(* CODESYS project SingleElevator_final.project

Project tree, tasks and I/O mapping:
  Device : CODESYS Control Win V3, 3S - Smart Software Solutions GmbH, version 3.5.15.40
    application Application
      libraries: Standard, * (System)
      task MainTask (cyclic, interval 100 ms, priority 1) calls Simulation, GA_collector, Policy
      task VISU_TASK (cyclic, interval 100 ms, priority 31) calls VisuElems.Visu_Prg
      global variables GVL
      visualisation Visualization
      program Simulation [ST]
      GAs/
        function block Door_module [SFC]: ready_active, busy_active, op_complete_active, reset_done_active, Init_active
        function block Cardinal [SFC]: Lights_active, Busy_active, Ready_active, Save_Arrays_active, Init_active, Cancel_call_active
        function block Moves_module [SFC]: G_floor_Problem_active, Stop_Op_Doors_down_active, Ready_active, Busy_active, Closing_Doors_active, Closing_Doors_exit, Init_active, Stop_Op_Doors_down_exit, Slow_d_active, Stop_Op_Doors_up_active, Slow_u_active, Fast_u_active, Stop_Op_Doors_up_exit, Check_Ramp_u_active, Check_Deck_u_active, Fast_d_active, Check_Ramp_d_active, Check_Deck_d_active, Stop_u_active, Stop_d_active, Errors_d_active, Errors_u_active, Homing_0_active, Homing_0_exit, Homing_1_active, Homing_2_active, Homing_3_active, Homing_3_exit, Exception_2_active, Exception_3_active, Exception_3_exit
      program GA_collector [FBD]
      program Policy [SFC]: Start_Cardinal_active, Error_routines_active, Start_Homing_active, Start_What_active, _aFinish_routine_active
  text list GlobalTextList
*)

// Device/Application/GVL
//{attribute 'qualified_only'}
VAR_GLOBAL
(* Elevator managing variables*)
	Open: BOOL;				(* Sensor: the door is fully open*)
	Closed: BOOL;			(* Sensor: the door is fully closed*)
	LimitDown: BOOL;		(* Sensor: lower limit sensor, if TRUE the lift has reached the lower limit*)
	LimitUp: BOOL;			(* Sensor: upper limit sensor, if TRUE the lift has reached the upper limit*)
	DeckSensor: BOOL;		(* Sensor: if TRUE the cab is in proximity of a deck*)
	RampSensor: BOOL;		(* Sensor: if TRUE the cab is in proximity of a ramp*)
	Presence :BOOL; 		(* Sensor: if TRUE something blocks the door photocell*)
	Emergency: BOOL;		(* Input: if TRUE the emergency button has been pressed*)

	Closing: BOOL;			(* Actuator: if TRUE the door starts closing*)
	Opening: BOOL;			(* Actuator: the door starts opening*)
	Motor_on: BOOL;			(* Actuator: if TRUE the lift pulley motor start moving*)
	Up: BOOL;				(* Actuator parameter: if TRUE the lift moves upward, downward otherwise*)
	Vel: BOOL;				(* Actuator parameter: motor speed, if TRUE high speed, low speed otherwise*)
	

	Current: INT;  			(* Visualization: variable used to storage the current deck*)
    Destination: INT;		(* Visualization: variable used to storage the the destination deck*)
	EmergencyVis: BOOL; 	(* Visualization: if TRUE the emergency light is turned on*)


	
	
	InitialDeck: INT := 1;	(* Only for simulation: variable used to define the initial deck*)
	InitCycle: BOOL := FALSE;(* Only for simulation: used to execute the instruction at the first cycle*)
	Height: INT;			(* Only for simulation: elevator height*)
	DeckRest: INT;        	(* Only for simulation: division rest for generating deck sensor*)
	Memory: INT;
	RampRest: INT;			(* Only for simulation: division rest for generating the ramp position*)
	MemoryR: INT;
	Door: INT;				(* Only for simulation: to visualize the closing of the door*)
	Displacement: INT;		(* Only for simulation: lift displacement, dependent on the motor speed*)

 (*Inputs: internal panel variables*)
	PG: BOOL;
	P1: BOOL;
	P2: BOOL;
	P3: BOOL;
	P4: BOOL;
	P5: BOOL;
	P6: BOOL;
	P7: BOOL;
	
	(*Inputs: external panel variables*)
	UpDeckG: BOOL;
	UpDeck1: BOOL;
	UpDeck2: BOOL;
	UpDeck3: BOOL;
	UpDeck4: BOOL;
	UpDeck5: BOOL;
	UpDeck6: BOOL;
	DownDeck7: BOOL;
	DownDeck6: BOOL;
	DownDeck5: BOOL;
	DownDeck4: BOOL;
	DownDeck3: BOOL;
	DownDeck2: BOOL;
	DownDeck1: BOOL;

(*Visualization: internal panel variables used to turn on the LED*)
	PGVis: BOOL;
	P1Vis: BOOL;
	P2Vis: BOOL;
	P3Vis: BOOL;
	P4Vis: BOOL;
	P5Vis: BOOL;
	P6Vis: BOOL;
	P7Vis: BOOL;

(*Visualization: external panel variables used to turn on the LED*)
	UpDeckGVis: BOOL;
	UpDeck1Vis: BOOL;
	UpDeck2Vis: BOOL;
	UpDeck3Vis: BOOL;
	UpDeck4Vis: BOOL;
	UpDeck5Vis: BOOL;
	UpDeck6Vis: BOOL;
	DownDeck7Vis: BOOL;
	DownDeck6Vis: BOOL;
	DownDeck5Vis: BOOL;
	DownDeck4Vis: BOOL;
	DownDeck3Vis: BOOL;
	DownDeck2Vis: BOOL;
	DownDeck1Vis: BOOL;

(*Only for simulation: variables used to simulate the fault on deck sensor*)
	SensorG: BOOL;				(* if TRUE the magnetic information for deck G is lost and the deck sensor cannot become TRUE*)
	Sensor1: BOOL;				(* if TRUE the magnetic information for deck 1 is lost and the deck sensor cannot become TRUE*)
	Sensor2: BOOL;
	Sensor3: BOOL;
	Sensor4: BOOL;
	Sensor5: BOOL;
	Sensor6: BOOL;
	Sensor7: BOOL;
	FaultSensorAlarm: BOOL; 	(* Visulaization: if TRUE alerts the user of a deck sensor fault*)

(*Only for simulation: variables used to simulate the fault on ramp sensor*)
	RampGUp: BOOL;
	Ramp1Down: BOOL;
	Ramp1Up:BOOL;
	Ramp2Down: BOOL;
	Ramp2Up:BOOL;
	Ramp3Down: BOOL;
	Ramp3Up:BOOL;
	Ramp4Down: BOOL;
	Ramp4Up:BOOL;
	Ramp5Down: BOOL;
	Ramp5Up:BOOL;
	Ramp6Down: BOOL;
	Ramp6Up:BOOL;
	Ramp7Down: BOOL;
	FaultRampAlarm: BOOL; 		(* Visulaization: if TRUE alerts the user of a ramp sensor fault*)
	SensorGOK: BOOL;
	Sensor1OK: BOOL;
	Sensor2OK: BOOL;
	Sensor6OK: BOOL;
	Sensor3OK: BOOL;
	Sensor4OK: BOOL;
	Sensor5OK: BOOL;
	Sensor7OK: BOOL;
	RampGUpOK: BOOL;
	Ramp1DownOK: BOOL;
	Ramp1UpOK: BOOL;
	Ramp2DownOK: BOOL;
	Ramp2UpOK: BOOL;
	Ramp3DownOK: BOOL;
	Ramp3UpOK: BOOL;
	Ramp4DownOK: BOOL;
	Ramp4UpOK: BOOL;
	Ramp5DownOK: BOOL;
	Ramp5UpOK: BOOL;
	Ramp6DownOK: BOOL;
	Ramp6UpOK: BOOL;
	Ramp7DownOK: BOOL;
	Ramp7UpOK: BOOL;
	
	//var aggiunte da me
	array_dest_up_onfly: ARRAY[0..7] OF INT;
	array_dest_up_stored: ARRAY[0..7] OF INT;
	
	array_dest_down_onfly: ARRAY[0..7] OF INT;
	array_dest_down_stored: ARRAY[0..7] OF INT;
	
	served_up: BOOL; // flag di fine servizio per movimento up
	served_down: BOOL; // flag di fine servizio per movimento down
	dest_target_up: INT; //destinazioen target up
	dest_target_down: INT; //destinazione target down
	enable_target_up_down: BOOL;	
	G_floor_problem: BOOL;
	
	//Istanze dei GA
	door_module_0: Door_module;
	Cardinal_0: Cardinal;
	Moves_module_0: Moves_module;

END_VAR

// Device/Application/Simulation
PROGRAM Simulation
VAR
END_VAR

(* Initial position of the cab inside the hoistway. It is executed only at the first cycle.  *)
IF NOT GVL.InitCycle THEN
			GVL.InitCycle := TRUE ;
			GVL.Height := 20 * GVL.InitialDeck;
		    GVL.Door := 0;
			GVL.Current := GVL.Height / 20;
END_IF;

(* Elevator management, these instructions are executed each cycle time*)

(* Elevator door control. *)
IF GVL.Closing THEN
	GVL.Door := GVL.Door + 1;		(*Closing door management*)
	GVL.Open := FALSE;
END_IF

IF GVL.Door >= 60 THEN						(* Closed door limit*)
	GVL.Closed := TRUE;
END_IF

IF GVL.Opening THEN
	GVL.Door := GVL.Door - 1; 	(* Opening door management*)
	GVL.Closed := FALSE;
END_IF

IF GVL.Door <= 0 THEN							(* Open door limit*)
	GVL.Open := TRUE;
END_IF


(* Maximum and minimum management in the door simulation*)
IF GVL.Door < 0 THEN
	 GVL.Door := 0;
END_IF

IF GVL.Door > 60 THEN
	GVL.Door := 60;
END_IF


(* Control of the cab position inside the hostway. *)
(* Displacement definition for graphic visualization*)
IF GVL.Vel THEN 
	GVL.Displacement := 2;
ELSE 
	GVL.Displacement := 1;
END_IF


(* Height modification relying on direction and speed*)
IF GVL.Motor_on AND GVL.Up THEN
	GVL.Height := GVL.Height + GVL.Displacement;
	GVL.LimitDown := FALSE;
END_IF

IF GVL.Motor_on AND NOT GVL.Up THEN
	GVL.Height := GVL.Height - GVL.Displacement;
	GVL.LimitUp := FALSE;
END_IF


(* Limits for visualization*)
IF GVL.Height < -20 THEN
	GVL.Height := -20;
END_IF

IF GVL.Height > 160 THEN
	GVL.Height := 160;
END_IF

(* Limit sensors management*)
IF GVL.Height <= -10 THEN
	GVL.LimitDown := TRUE;
END_IF

IF GVL.Height >= 150 THEN
	 GVL.LimitUp := TRUE;
END_IF


(*-------------------------------------------------------------------*)
(*  Fault Management (Deck and Ramp Sensors)   *)
(*-------------------------------------------------------------------*)
(* Deck Sensor*)
(* Range of value where the deck sensor is active*)
IF ((GVL.Height >= -1) AND (GVL.Height <= 1)) THEN
	GVL.SensorGOK := TRUE;
ELSE  
	GVL.SensorGOK := FALSE;
END_IF

IF ((GVL.Height >= 20-1) AND (GVL.Height <= 20+1)) THEN
	GVL.Sensor1OK := TRUE;
ELSE  
	GVL.Sensor1OK := FALSE;
END_IF

IF ((GVL.Height >= 40-1) AND (GVL.Height <= 40+1)) THEN
	GVL.Sensor2OK := TRUE;
ELSE  
	GVL.Sensor2OK := FALSE;
END_IF

IF ((GVL.Height >= 60-1) AND (GVL.Height <= 60+1)) THEN
	GVL.Sensor3OK := TRUE;
ELSE  
	GVL.Sensor3OK := FALSE;
END_IF

IF ((GVL.Height >= 80-1) AND (GVL.Height <= 80+1)) THEN
	GVL.Sensor4OK := TRUE;
ELSE  
	GVL.Sensor4OK := FALSE;
END_IF

IF ((GVL.Height >= 100-1) AND (GVL.Height <= 100+1)) THEN
	GVL.Sensor5OK := TRUE;
ELSE   
	GVL.Sensor5OK := FALSE;
END_IF

IF ((GVL.Height >= 120-1) AND (GVL.Height <= 120+1)) THEN
	GVL.Sensor6OK := TRUE;
ELSE  
	GVL.Sensor6OK := FALSE;
END_IF

IF ((GVL.Height >= 140-1) AND (GVL.Height <= 140+1)) THEN
	GVL.Sensor7OK := TRUE;
ELSE  
	GVL.Sensor7OK := FALSE;
END_IF

GVL.DeckSensor := (GVL.SensorGOK AND NOT GVL.SensorG) OR
				    (GVL.Sensor1OK AND NOT GVL.Sensor1) OR
				    (GVL.Sensor2OK AND NOT GVL.Sensor2) OR
				    (GVL.Sensor3OK AND NOT GVL.Sensor3) OR
				    (GVL.Sensor4OK AND NOT GVL.Sensor4) OR
				    (GVL.Sensor5OK AND NOT GVL.Sensor5) OR
				    (GVL.Sensor6OK AND NOT GVL.Sensor6) OR
				    (GVL.Sensor7OK AND NOT GVL.Sensor7);

(* Ramp Sensor*)
(* Range of value where the ramp sensor is active*)
IF ((GVL.Height >= 5-1) AND (GVL.Height <= 5+1)) THEN
	GVL.RampGUpOK := TRUE;
ELSE 
	GVL.RampGUpOK := FALSE;
END_IF

(* Ramp close to deck 1*)
IF ((GVL.Height >= 15-1) AND (GVL.Height <= 15+1)) THEN
	GVL.Ramp1DownOK := TRUE;
ELSE 
	GVL.Ramp1DownOK := FALSE;
END_IF

IF ((GVL.Height >= 25-1) AND (GVL.Height <= 25+1)) THEN
	GVL.Ramp1UpOK := TRUE;
ELSE 
	GVL.Ramp1UpOK := FALSE;
END_IF

(* Ramp close to deck 2*)
IF ((GVL.Height >= 35-1) AND (GVL.Height <= 35+1)) THEN
	GVL.Ramp2DownOK := TRUE;
ELSE 
	GVL.Ramp2DownOK := FALSE;
END_IF

IF ((GVL.Height >= 45-1) AND (GVL.Height <= 45+1)) THEN
	GVL.Ramp2UpOK := TRUE;
ELSE 
	GVL.Ramp2UpOK := FALSE;
END_IF

(*Ramp close to deck  3*)
IF ((GVL.Height >= 55-1) AND (GVL.Height <= 55+1)) THEN
	GVL.Ramp3DownOK := TRUE;
ELSE 
	GVL.Ramp3DownOK := FALSE;
END_IF

IF ((GVL.Height >= 65-1) AND (GVL.Height <= 65+1)) THEN
	GVL.Ramp3UpOK := TRUE;
ELSE 
	GVL.Ramp3UpOK := FALSE;
END_IF

(* Ramp close to deck  4*)
IF ((GVL.Height >= 75-1) AND (GVL.Height <= 75+1)) THEN
	GVL.Ramp4DownOK := TRUE;
ELSE 
	GVL.Ramp4DownOK := FALSE;
END_IF

IF ((GVL.Height >= 85-1) AND (GVL.Height <= 85+1)) THEN
	GVL.Ramp4UpOK := TRUE;
ELSE 
	GVL.Ramp4UpOK:=FALSE;
END_IF

(* Ramp close to deck  5*)
IF ((GVL.Height >= 95-1) AND (GVL.Height <= 95+1)) THEN
	GVL.Ramp5DownOK := TRUE;
ELSE 
	GVL.Ramp5DownOK := FALSE;
END_IF

IF ((GVL.Height >= 105-1) AND (GVL.Height <= 105+1)) THEN
	GVL.Ramp5UpOK := TRUE;
ELSE
	GVL.Ramp5UpOK := FALSE;
END_IF

(* Ramp close to deck  6*)
IF ((GVL.Height >= 115-1) AND (GVL.Height <= 115+1)) THEN
	GVL.Ramp6DownOK := TRUE;
ELSE 
	GVL.Ramp6DownOK := FALSE;
END_IF

IF ((GVL.Height >= 125-1) AND (GVL.Height <= 125+1)) THEN
	GVL.Ramp6UpOK := TRUE;
ELSE 
	GVL.Ramp6UpOK := FALSE;
END_IF

(* Ramp close to deck  7*)
IF ((GVL.Height >= 135-1) AND (GVL.Height <= 135+1)) THEN
	GVL.Ramp7DownOK := TRUE;
ELSE 
	GVL.Ramp7DownOK := FALSE;
END_IF

GVL.RampSensor:=(GVL.RampGUpOK AND NOT GVL.RampGUp) OR 
								(GVL.Ramp1DownOK AND NOT GVL.Ramp1Down ) OR 
								(GVL.Ramp1UpOK AND NOT GVL.Ramp1Up ) OR
								(GVL.Ramp2DownOK AND NOT GVL.Ramp2Down ) OR 
								(GVL.Ramp2UpOK AND NOT GVL.Ramp2Up ) OR
								(GVL.Ramp3DownOK AND NOT GVL.Ramp3Down ) OR
 								(GVL.Ramp3UpOK AND NOT GVL.Ramp3Up ) OR
								(GVL.Ramp4DownOK AND NOT GVL.Ramp4Down ) OR
 								(GVL.Ramp4UpOK AND NOT GVL.Ramp4Up ) OR
								(GVL.Ramp5DownOK AND NOT GVL.Ramp5Down ) OR
 								(GVL.Ramp5UpOK AND NOT GVL.Ramp5Up ) OR
								(GVL.Ramp6DownOK AND NOT GVL.Ramp6Down ) OR
								(GVL.Ramp6UpOK AND NOT GVL.Ramp6Up ) OR
								(GVL.Ramp7DownOK AND NOT GVL.Ramp7Down );

END_PROGRAM

// Device/Application/GA_collector
PROGRAM GA_collector
VAR



END_VAR

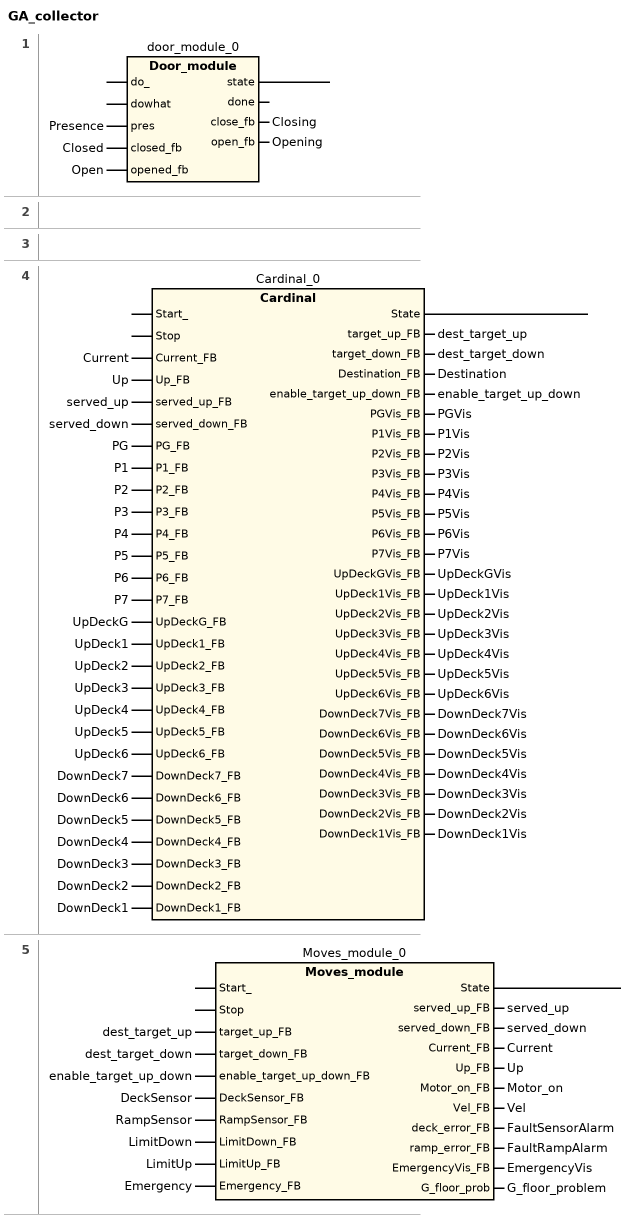
// NETWORK 1
door_module_0(
    pres := Presence,
    closed_fb := Closed,
    opened_fb := Open,
    close_fb => Closing,
    open_fb => Opening); // Door_module

// NETWORK 2

// NETWORK 3

// NETWORK 4
Cardinal_0(
    Current_FB := Current,
    Up_FB := Up,
    served_up_FB := served_up,
    served_down_FB := served_down,
    PG_FB := PG,
    P1_FB := P1,
    P2_FB := P2,
    P3_FB := P3,
    P4_FB := P4,
    P5_FB := P5,
    P6_FB := P6,
    P7_FB := P7,
    UpDeckG_FB := UpDeckG,
    UpDeck1_FB := UpDeck1,
    UpDeck2_FB := UpDeck2,
    UpDeck3_FB := UpDeck3,
    UpDeck4_FB := UpDeck4,
    UpDeck5_FB := UpDeck5,
    UpDeck6_FB := UpDeck6,
    DownDeck7_FB := DownDeck7,
    DownDeck6_FB := DownDeck6,
    DownDeck5_FB := DownDeck5,
    DownDeck4_FB := DownDeck4,
    DownDeck3_FB := DownDeck3,
    DownDeck2_FB := DownDeck2,
    DownDeck1_FB := DownDeck1,
    target_up_FB => dest_target_up,
    target_down_FB => dest_target_down,
    Destination_FB => Destination,
    enable_target_up_down_FB => enable_target_up_down,
    PGVis_FB => PGVis,
    P1Vis_FB => P1Vis,
    P2Vis_FB => P2Vis,
    P3Vis_FB => P3Vis,
    P4Vis_FB => P4Vis,
    P5Vis_FB => P5Vis,
    P6Vis_FB => P6Vis,
    P7Vis_FB => P7Vis,
    UpDeckGVis_FB => UpDeckGVis,
    UpDeck1Vis_FB => UpDeck1Vis,
    UpDeck2Vis_FB => UpDeck2Vis,
    UpDeck3Vis_FB => UpDeck3Vis,
    UpDeck4Vis_FB => UpDeck4Vis,
    UpDeck5Vis_FB => UpDeck5Vis,
    UpDeck6Vis_FB => UpDeck6Vis,
    DownDeck7Vis_FB => DownDeck7Vis,
    DownDeck6Vis_FB => DownDeck6Vis,
    DownDeck5Vis_FB => DownDeck5Vis,
    DownDeck4Vis_FB => DownDeck4Vis,
    DownDeck3Vis_FB => DownDeck3Vis,
    DownDeck2Vis_FB => DownDeck2Vis,
    DownDeck1Vis_FB => DownDeck1Vis); // Cardinal

// NETWORK 5
Moves_module_0(
    target_up_FB := dest_target_up,
    target_down_FB := dest_target_down,
    enable_target_up_down_FB := enable_target_up_down,
    DeckSensor_FB := DeckSensor,
    RampSensor_FB := RampSensor,
    LimitDown_FB := LimitDown,
    LimitUp_FB := LimitUp,
    Emergency_FB := Emergency,
    served_up_FB => served_up,
    served_down_FB => served_down,
    Current_FB => Current,
    Up_FB => Up,
    Motor_on_FB => Motor_on,
    Vel_FB => Vel,
    deck_error_FB => FaultSensorAlarm,
    ramp_error_FB => FaultRampAlarm,
    EmergencyVis_FB => EmergencyVis,
    G_floor_prob => G_floor_problem); // Moves_module

END_PROGRAM

// Device/Application/GAs/Door_module
FUNCTION_BLOCK Door_module
VAR_INPUT
	do_: BOOL;
	dowhat: STRING;
	pres: BOOL;
	closed_fb: BOOL;
	opened_fb: BOOL;
END_VAR
VAR_OUTPUT
	state: STRING;
	done: BOOL;
	close_fb: BOOL;
	open_fb: BOOL;
END_VAR
VAR
END_VAR

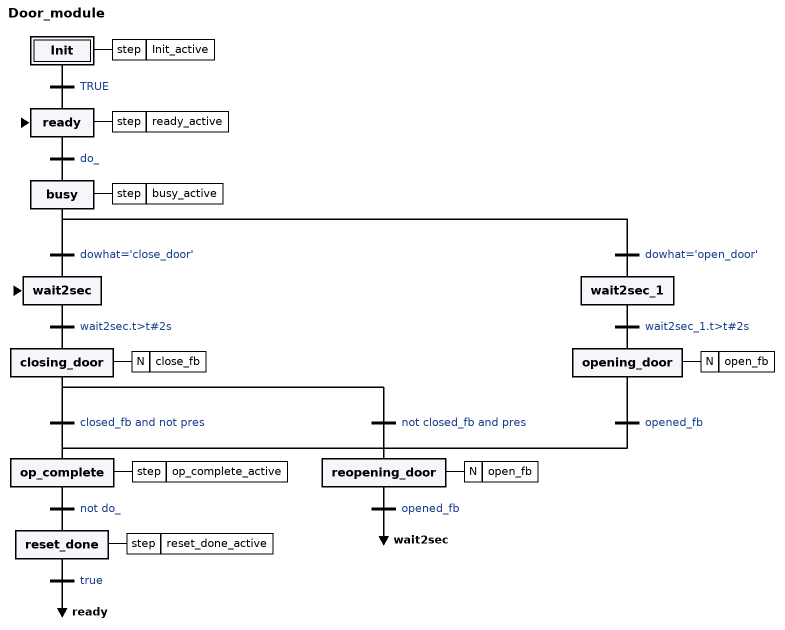
INITIAL_STEP Init:
    Init_active(N);  // step action
END_STEP
TRANSITION FROM Init TO ready
    := TRUE;
END_TRANSITION
STEP ready:
    ready_active(N);  // step action
END_STEP
TRANSITION FROM ready TO busy
    := do_;
END_TRANSITION
STEP busy:
    busy_active(N);  // step action
END_STEP
TRANSITION FROM busy TO wait2sec
    := dowhat='close_door';
END_TRANSITION
STEP wait2sec:
END_STEP
TRANSITION FROM wait2sec TO closing_door
    := wait2sec.t>t#2s;
END_TRANSITION
STEP closing_door:
    close_fb(N);
END_STEP
TRANSITION FROM closing_door TO op_complete
    := closed_fb and not pres;
END_TRANSITION
TRANSITION FROM closing_door TO reopening_door
    := not closed_fb and pres;
END_TRANSITION
STEP reopening_door:
    open_fb(N);
END_STEP
TRANSITION FROM reopening_door TO wait2sec
    := opened_fb;
END_TRANSITION
TRANSITION FROM busy TO wait2sec_1
    := dowhat='open_door';
END_TRANSITION
STEP wait2sec_1:
END_STEP
TRANSITION FROM wait2sec_1 TO opening_door
    := wait2sec_1.t>t#2s;
END_TRANSITION
STEP opening_door:
    open_fb(N);
END_STEP
TRANSITION FROM opening_door TO op_complete
    := opened_fb;
END_TRANSITION
STEP op_complete:
    op_complete_active(N);  // step action
END_STEP
TRANSITION FROM op_complete TO reset_done
    := not do_;
END_TRANSITION
STEP reset_done:
    reset_done_active(N);  // step action
END_STEP
TRANSITION FROM reset_done TO ready
    := true;
END_TRANSITION

ACTION ready_active:
state:='ready';
END_ACTION

ACTION busy_active:
state:='busy';
END_ACTION

ACTION op_complete_active:
done:=TRUE;
END_ACTION

ACTION reset_done_active:
done:=FALSE;
END_ACTION

ACTION Init_active:
//INZIALIZZAZIONE DEGLI OUTPUT DI DOOR_MODULE
done:=FALSE;
close_fb:=FALSE;
open_fb:=FALSE;
END_ACTION

END_FUNCTION_BLOCK

// Device/Application/GAs/Cardinal
FUNCTION_BLOCK Cardinal
VAR_INPUT
	
	Start_: BOOL;
	Stop: BOOL;
	Current_FB: INT; //visualizzazione piano corrente	

	Up_FB:BOOL;
	
	served_up_FB: BOOL; // flag di finito servizio del valore target_up
	served_down_FB: BOOL; // flag di finito servizio del valore target_down
	
	 (*Inputs: internal panel variables*)
	PG_FB: BOOL;
	P1_FB: BOOL;
	P2_FB: BOOL;
	P3_FB: BOOL;
	P4_FB: BOOL;
	P5_FB: BOOL;
	P6_FB: BOOL;
	P7_FB: BOOL;
	
	(*Inputs: external panel variables*)
	UpDeckG_FB: BOOL;
	UpDeck1_FB: BOOL;
	UpDeck2_FB: BOOL;
	UpDeck3_FB: BOOL;
	UpDeck4_FB: BOOL;
	UpDeck5_FB: BOOL;
	UpDeck6_FB: BOOL;
	DownDeck7_FB: BOOL;
	DownDeck6_FB: BOOL;
	DownDeck5_FB: BOOL;
	DownDeck4_FB: BOOL;
	DownDeck3_FB: BOOL;
	DownDeck2_FB: BOOL;
	DownDeck1_FB: BOOL;
END_VAR
VAR_OUTPUT
	
	State: STRING;
	
	target_up_FB: INT; // valore da dare a Dest_target_up
	target_down_FB: INT; // valore da dare a Dest_target_down
	
	Destination_FB: INT; //visualizzazione del piano destinazione
	
	enable_target_up_down_FB: BOOL; //per manovrare in moves_module il verso di percorrenza
	
(*Visualization: internal panel variables used to turn on the LED*)
	PGVis_FB: BOOL;
	P1Vis_FB: BOOL;
	P2Vis_FB: BOOL;
	P3Vis_FB: BOOL;
	P4Vis_FB: BOOL;
	P5Vis_FB: BOOL;
	P6Vis_FB: BOOL;
	P7Vis_FB: BOOL;

(*Visualization: external panel variables used to turn on the LED*)
	UpDeckGVis_FB: BOOL;
	UpDeck1Vis_FB: BOOL;
	UpDeck2Vis_FB: BOOL;
	UpDeck3Vis_FB: BOOL;
	UpDeck4Vis_FB: BOOL;
	UpDeck5Vis_FB: BOOL;
	UpDeck6Vis_FB: BOOL;
	DownDeck7Vis_FB: BOOL;
	DownDeck6Vis_FB: BOOL;
	DownDeck5Vis_FB: BOOL;
	DownDeck4Vis_FB: BOOL;
	DownDeck3Vis_FB: BOOL;
	DownDeck2Vis_FB: BOOL;
	DownDeck1Vis_FB: BOOL;
	
END_VAR
VAR
	Dest_floor: INT;//contiene variabile destinazione
	can_be_clicked: BOOL;
	up_motion: BOOL; 
	prio: INT;

	//ARRAY DELLE CHIAMATE

	array_dest_up_onfly_FB: ARRAY[0..7] OF INT;

	array_dest_up_stored_FB: ARRAY[0..7] OF INT;
	

	array_dest_down_onfly_FB: ARRAY[0..7] OF INT;

	array_dest_down_stored_FB: ARRAY[0..7] OF INT;
	
	// contatori di scorrimento per la scrittura degli array,
	sliding_index_1: INT;
	sliding_index_2: INT;
	sliding_index_3: INT;
	sliding_index_4: INT;
	
	// contatori di riordino array
	k: INT;
	i: INT;
	k_1: INT;
	i_1: INT;

	//variabili appoggio riordino array
	var1: INT;

	var1_1: INT;
	
	min_index: INT;
	min_index_1: INT;
	max_index: INT;
	max_index_1: INT;
	already_pres: BOOL;

	//contatori generici 	
	counter_calls_up_stored: INT;
	counter_calls_down_stored: INT;
	counter_calls_up_onfly: INT;
	counter_calls_down_onfly: INT;

	cont: INT;
	cancel_time: BOOL;
END_VAR

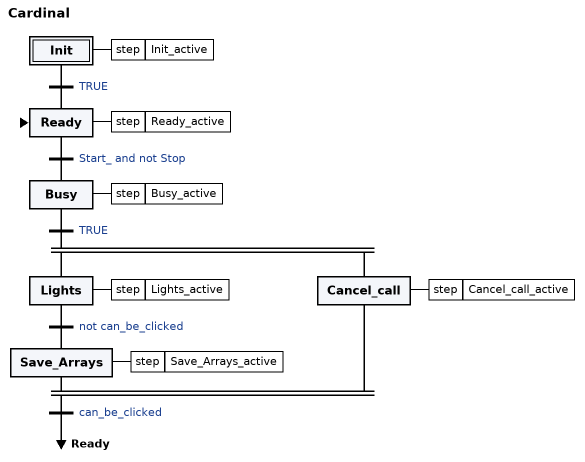
INITIAL_STEP Init:
    Init_active(N);  // step action
END_STEP
TRANSITION FROM Init TO Ready
    := TRUE;
END_TRANSITION
STEP Ready:
    Ready_active(N);  // step action
END_STEP
TRANSITION FROM Ready TO Busy
    := Start_ and not Stop;
END_TRANSITION
STEP Busy:
    Busy_active(N);  // step action
END_STEP
TRANSITION FROM Busy TO (Lights, Cancel_call)
    := TRUE;
END_TRANSITION
STEP Lights:
    Lights_active(N);  // step action
END_STEP
TRANSITION FROM Lights TO Save_Arrays
    := not can_be_clicked;
END_TRANSITION
STEP Save_Arrays:
    Save_Arrays_active(N);  // step action
END_STEP
STEP Cancel_call:
    Cancel_call_active(N);  // step action
END_STEP
TRANSITION FROM (Save_Arrays, Cancel_call) TO Ready
    := can_be_clicked;
END_TRANSITION

ACTION Lights_active:
//INTERFACCIAMENTO CON LE CHIAMATE DA PULSANTIERA INTERNA
(*
HO SCELTO DI DARE A QUESTE CHIAMATE UN 'VERSO' IN MODO DA TRATTARLE ALLO STESSO MODO DELLE CHIAMATE
DA PULSANTIERA ESTERNA, IL VERSO IN QUESTIONE DERIVA DAL FLAG up_elev_curr_FB CHE DERIVA DAL FLAG
DEL VERSO DELL'ASCENSORE IN USCITA DAL GA DI MOVIMENTO (MOVES_MODULE) CON VALORE AD INIZIO PROGRAMMA
PARI A TRUE PERCHE DOPO L'HOMING POSSO SOLO ANDARE IN ALTO. E' UN PRINCIPIO DI RETROAZIONE PERCHE A 
SUA VOLTA MOVES_MODULE LEGGERA' LE USCITE DI CARDINAL PER SAPERE LA DESTINAZIONE.
*)

//up_elev_curr_FB: FLAG IN INGRESSO AL CARDINAL E IN OUTPUT A MOVES_MODULE
//up_motion: VIENE LETTO DOPO PER SAPERE DOVE SMISTARE LE CALLS

IF PG_FB AND can_be_clicked THEN
	PGVis_FB:=TRUE;
	can_be_clicked:=FALSE;
	Dest_floor:=0;
	IF Dest_floor>Current_FB THEN
		up_motion:=TRUE;
	ELSE
		up_motion:=FALSE;
	END_IF
END_IF
IF P1_FB AND can_be_clicked THEN
	P1Vis_FB:=TRUE;
	can_be_clicked:=FALSE;
	Dest_floor:=1;
	IF Dest_floor>Current_FB THEN
		up_motion:=TRUE;
	ELSE
		up_motion:=FALSE;
	END_IF
END_IF
IF P2_FB AND can_be_clicked  THEN
	P2Vis_FB:=TRUE;
	can_be_clicked:=FALSE;
	Dest_floor:=2;
	IF Dest_floor>Current_FB THEN
		up_motion:=TRUE;
	ELSE
		up_motion:=FALSE;
	END_IF
END_IF
IF P3_FB AND can_be_clicked  THEN
	P3Vis_FB:=TRUE;
	can_be_clicked:=FALSE;
	Dest_floor:=3;
	IF Dest_floor>Current_FB THEN
		up_motion:=TRUE;
	ELSE
		up_motion:=FALSE;
	END_IF
END_IF
IF P4_FB AND can_be_clicked  THEN
	P4Vis_FB:=TRUE;
	can_be_clicked:=FALSE;
	Dest_floor:=4;
	IF Dest_floor>Current_FB THEN
		up_motion:=TRUE;
	ELSE
		up_motion:=FALSE;
	END_IF
END_IF
IF P5_FB AND can_be_clicked  THEN
	P5Vis_FB:=TRUE;
	can_be_clicked:=FALSE;
	Dest_floor:=5;
	IF Dest_floor>Current_FB THEN
		up_motion:=TRUE;
	ELSE
		up_motion:=FALSE;
	END_IF
END_IF
IF P6_FB AND can_be_clicked  THEN
	P6Vis_FB:=TRUE;
	can_be_clicked:=FALSE;
	Dest_floor:=6;
	IF Dest_floor>Current_FB THEN
		up_motion:=TRUE;
	ELSE
		up_motion:=FALSE;
	END_IF
END_IF
IF P7_FB AND can_be_clicked  THEN
	P7Vis_FB:=TRUE;
	can_be_clicked:=FALSE;
	Dest_floor:=7;
	IF Dest_floor>Current_FB THEN
		up_motion:=TRUE;
	ELSE
		up_motion:=FALSE;
	END_IF
END_IF

//INTERFACCIAMENTO CON LE PULSANTIERE ESTERNE

(*QUI IL VERSO DELLA CHIAMATA INVECE E' FISSATO*)

IF UpDeckG_FB AND can_be_clicked  THEN
	UpDeckGVis_FB:=TRUE;
	can_be_clicked:=FALSE;
	Dest_floor:=0;
	up_motion:=TRUE;
END_IF
IF UpDeck1_FB AND can_be_clicked  THEN
	UpDeck1Vis_FB:=TRUE;
	can_be_clicked:=FALSE;
	Dest_floor:=1;
	up_motion:=TRUE;
END_IF
IF UpDeck2_FB AND can_be_clicked  THEN
	UpDeck2Vis_FB:=TRUE;
	can_be_clicked:=FALSE;
	Dest_floor:=2;
	up_motion:=TRUE;
END_IF
IF UpDeck3_FB AND can_be_clicked  THEN
	UpDeck3Vis_FB:=TRUE;
	can_be_clicked:=FALSE;
	Dest_floor:=3;
	up_motion:=TRUE;
END_IF
IF UpDeck4_FB AND can_be_clicked  THEN
	UpDeck4Vis_FB:=TRUE;
	can_be_clicked:=FALSE;
	Dest_floor:=4;
	up_motion:=TRUE;
END_IF
IF UpDeck5_FB AND can_be_clicked  THEN
	UpDeck5Vis_FB:=TRUE;
	can_be_clicked:=FALSE;
	Dest_floor:=5;
	up_motion:=TRUE;
END_IF
IF UpDeck6_FB AND can_be_clicked  THEN
	UpDeck6Vis_FB:=TRUE;
	can_be_clicked:=FALSE;
	Dest_floor:=6;
	up_motion:=TRUE;
END_IF
IF DownDeck7_FB AND can_be_clicked  THEN
	DownDeck7Vis_FB:=TRUE;
	can_be_clicked:=FALSE;
	Dest_floor:=7;
	up_motion:=FALSE;
END_IF
IF DownDeck6_FB AND can_be_clicked  THEN
	DownDeck6Vis_FB:=TRUE;
	can_be_clicked:=FALSE;
	Dest_floor:=6;
	up_motion:=FALSE;
END_IF
IF DownDeck5_FB AND can_be_clicked  THEN
 	DownDeck5Vis_FB:=TRUE;
	can_be_clicked:=FALSE;
	Dest_floor:=5;
	up_motion:=FALSE;
END_IF
IF DownDeck4_FB AND can_be_clicked  THEN
	DownDeck4Vis_FB:=TRUE;
	can_be_clicked:=FALSE;
	Dest_floor:=4;
	up_motion:=FALSE;
END_IF
IF DownDeck3_FB AND can_be_clicked  THEN
	DownDeck3Vis_FB:=TRUE;
	can_be_clicked:=FALSE;
	Dest_floor:=3;
	up_motion:=FALSE;
END_IF
IF DownDeck2_FB AND can_be_clicked  THEN
	DownDeck2Vis_FB:=TRUE;
	can_be_clicked:=FALSE;
	Dest_floor:=2;
	up_motion:=FALSE;
END_IF
IF DownDeck1_FB AND can_be_clicked  THEN
	DownDeck1Vis_FB:=TRUE;
	can_be_clicked:=FALSE;
	Dest_floor:=1;
	up_motion:=FALSE;
END_IF
END_ACTION

ACTION Busy_active:
State:='busy';
END_ACTION

ACTION Ready_active:
State:='ready';
END_ACTION

ACTION Save_Arrays_active:
//ARRAY_UP 
IF up_motion THEN
	FOR i := 0 TO 7 BY 1 DO
		IF Dest_floor=array_dest_up_onfly_FB[i] THEN
			already_pres:=TRUE;
		END_IF
	END_FOR
	IF NOT already_pres THEN
//VADO NELL'ARRAY DELLE CHIAMATE ONLFLY	
		IF Dest_floor>Current_FB THEN //vado negli array per le chiamate onfly
			array_dest_up_onfly_FB[sliding_index_1]:= Dest_floor; // carico nell'array delle dest
			sliding_index_1:=sliding_index_1+1; // incremento l'indice entro cui metterò la prossima chiamata verso l'alto 
			k:=0;
			i:=0;
			//PARTO CON L'ORDINAMENTO CON IL SELECTION SORTER
			WHILE i<=7 DO
				k:=i+1;
				min_index:=i;
				WHILE k<=7 DO
					IF array_dest_up_onfly_FB[k]<array_dest_up_onfly_FB[i] THEN
						min_index:=k;
					END_IF	
					k:=k+1;
				END_WHILE
				var1:= array_dest_up_onfly_FB[i];	
				array_dest_up_onfly_FB[i]:=array_dest_up_onfly_FB[min_index];	
				array_dest_up_onfly_FB[min_index]:=var1;
				i:=i+1;
			END_WHILE
		ELSIF Dest_floor<=Current_FB THEN
//VADO NELL'ARRAY DELLE CHIAMATE STORED			
			array_dest_up_stored_FB[sliding_index_2]:= Dest_floor; // carico nell'array delle dest
			sliding_index_2:=sliding_index_2+1; // incremento l'indice entro cui metterò la prossima chiamata verso l'alto
			k:=0;
			i:=0;
			//PARTO CON L'ORDINAMENTO CON IL SELECTION SORTER
			WHILE i<=7 DO
				k:=i+1;
				min_index:=i;
				WHILE k<=7 DO
					IF array_dest_up_stored_FB[k]<array_dest_up_stored_FB[i] THEN
						min_index:=k;
					END_IF	
					k:=k+1;
				END_WHILE
				var1:= array_dest_up_stored_FB[i];
				array_dest_up_stored_FB[i]:=array_dest_up_stored_FB[min_index];	
				array_dest_up_stored_FB[min_index]:=var1;
				i:=i+1;
			END_WHILE
		END_IF
	target_up_FB:=array_dest_up_onfly_FB[0];
	END_IF
	IF target_up_FB=8 THEN
//CONTROLLO IL PRIMO VALORE DELL'ARRAY UP, SE=8 PROVO A VEDERE GLI ALTRI ARRAY	
		FOR cont := 0 TO 7 BY 1 DO
			IF array_dest_up_onfly_FB[cont]=8 THEN
				counter_calls_up_onfly:= counter_calls_up_onfly+1;
			END_IF
			IF array_dest_down_onfly_FB[cont]=-1 THEN
				counter_calls_down_onfly:= counter_calls_down_onfly+1;
			END_IF
			IF array_dest_up_stored_FB[cont]=8 THEN
				counter_calls_up_stored:= counter_calls_up_stored+1;
			END_IF
			IF array_dest_down_stored_FB[cont]=-1 THEN
				counter_calls_down_stored:= counter_calls_down_stored+1;
			END_IF
		END_FOR
//ORA PROCEDO ALLE CASISTICHE
(*CASO CON:
FLY_UP VUOTO
FLY_DOWN PIENO
STORED_UP INDIFFERENTE
STORED_DOWN INDIFFERENTE
COPIO LE CHIAMATE STORED_UP IN FLY_UP MENTRE SERVO FLY_DOWN
 *)
		IF 	counter_calls_up_onfly=8 AND counter_calls_down_onfly<8 AND 
			counter_calls_up_stored<=8 AND counter_calls_down_stored<=8 THEN	

			FOR cont := 0 TO 7 BY 1 DO
				array_dest_up_onfly_FB[cont]:=array_dest_up_stored_FB[cont];
				array_dest_up_stored_FB[cont]:=8;
			END_FOR;
			sliding_index_1:=sliding_index_2;
			sliding_index_2:=0;
			enable_target_up_down_FB:=FALSE; //INVERSIONE DI MOTO VERSO IL BASSO
		END_IF
(*CASO CON:
FLY_UP VUOTO
FLY_DOWN VUOTO
STORED_UP PIENO
STORED_DOWN VUOTO
COPIO LA PRIMA CALL IN FLY_DOWN E LE ALTRE IN FLY_UP, IN MODO CHE POSSA TORNARE GIù FINO ALLA 
CALL CON DESTINAZIONE MINORE
*)
		IF 	counter_calls_up_onfly=8 AND counter_calls_down_onfly=8 AND 
			counter_calls_up_stored<8 AND counter_calls_down_stored=8 THEN
//in prova		
			array_dest_down_onfly_FB[0]:=array_dest_up_stored_FB[0];
			FOR cont := 1 TO 7 BY 1 DO
				array_dest_up_onfly_FB[cont]:=array_dest_up_stored_FB[cont];
				array_dest_up_stored_FB[cont]:=8;
			END_FOR;
			sliding_index_1:=sliding_index_2-1;
			sliding_index_2:=0;
			sliding_index_3:=1;
			enable_target_up_down_FB:=FALSE;
		END_IF
	ELSE
		enable_target_up_down_FB:=TRUE;
	END_IF
	
	can_be_clicked:=TRUE;
//ARRAY_DOWN
ELSE
	FOR i := 0 TO 7 BY 1 DO
		IF Dest_floor=array_dest_down_onfly_FB[i] THEN
			already_pres:=TRUE;
		END_IF
	END_FOR
	IF NOT already_pres THEN
//VADO NELL'ARRAY DELLE CHIAMATE ONLFLY
		IF Dest_floor<Current_FB  THEN
			array_dest_down_onfly_FB[sliding_index_3]:= Dest_floor; // carico nell'array delle dest
			sliding_index_3:=sliding_index_3+1; // incremento l'indice entro cui metterò la prossima chiamata verso l'alto 
			k:=0;
			i:=0;
//PARTO CON L'ORDINAMENTO CON IL SELECTION SORTER
			WHILE i<=7 DO
				k:=i+1;
				max_index:=i;
				WHILE k<=7 DO
					IF array_dest_down_onfly_FB[k]>array_dest_down_onfly_FB[i] THEN
						max_index:=k;
					END_IF
					k:=k+1;
				END_WHILE
				var1:= array_dest_down_onfly_FB[i];
				array_dest_down_onfly_FB[i]:=array_dest_down_onfly_FB[max_index];
				array_dest_down_onfly_FB[max_index]:=var1;	
				i:=i+1;
			END_WHILE
		ELSIF Dest_floor>=Current_FB THEN
//VADO NEGLI ARRAY PER LE CHIAMTE STORED
			array_dest_down_stored_FB[sliding_index_4]:= Dest_floor; // carico nell'array delle dest
			sliding_index_4:=sliding_index_4+1; // incremento l'indice entro cui metterò la prossima chiamata verso l'alto
			k:=0;
			i:=0;
//PARTO CON L'ORDINAMENTO CON IL SELECTION SORTER
			WHILE i<=7 DO
				k:=i+1;
				max_index:=i;
				WHILE k<=7 DO
					IF array_dest_down_stored_FB[i]<array_dest_down_stored_FB[k] THEN
						max_index:=k;
					END_IF	
					k:=k+1;
				END_WHILE
				var1:= array_dest_down_stored_FB[i];
				array_dest_down_stored_FB[i]:=array_dest_down_stored_FB[max_index];
				array_dest_down_stored_FB[max_index]:=var1;
				i:=i+1;
			END_WHILE
		END_IF
	target_down_FB:=array_dest_down_onfly_FB[0];
	END_IF
	IF target_down_FB=-1 THEN
//CONTROLLO IL PRIMO VALORE DELL'ARRAY UP, SE=8 PROVO A VEDERE GLI ALTRI ARRAY	
		FOR cont := 0 TO 7 BY 1 DO
			IF array_dest_up_onfly_FB[cont]=8 THEN
				counter_calls_up_onfly:= counter_calls_up_onfly+1;
			END_IF
			IF array_dest_down_onfly_FB[cont]=-1 THEN
				counter_calls_down_onfly:= counter_calls_down_onfly+1;
			END_IF
			IF array_dest_up_stored_FB[cont]=8 THEN
				counter_calls_up_stored:= counter_calls_up_stored+1;
			END_IF
			IF array_dest_down_stored_FB[cont]=-1 THEN
				counter_calls_down_stored:= counter_calls_down_stored+1;
			END_IF
		END_FOR
//ORA PROCEDO ALLE CASISTICHE
(*CASO CON:
FLY_UP PIENO
FLY_DOWN VUOTO
STORED_UP INDIFFERENTE
STORED_DOWN INDIFFERENTE
COPIO LE CHIAMATE STORED_DOWN IN FLY_DOWN MENTRE SERVO FLY_UP
 *)
		IF 	counter_calls_up_onfly<8 AND counter_calls_down_onfly=8 AND 
			counter_calls_up_stored<=8 AND counter_calls_down_stored<=8 THEN	

			FOR cont := 0 TO 7 BY 1 DO
				array_dest_down_onfly_FB[cont]:=array_dest_down_stored_FB[cont];
				array_dest_down_stored_FB[cont]:=-1;
			END_FOR;
			sliding_index_3:=sliding_index_4;
			sliding_index_4:=0;
			enable_target_up_down_FB:=TRUE;
		END_IF
(*CASO CON:
FLY_UP VUOTO
FLY_DOWN VUOTO
STORED_UP VUOTO
STORED_DOWN PIENO
COPIO LA PRIMA CALL IN FLY_UP E LE ALTRE IN FLY_DOWN, IN MODO CHE POSSA TORNARE SU FINO ALLA 
CALL CON DESTINAZIONE MAGGIORE
*)
		IF 	counter_calls_up_onfly=8 AND counter_calls_down_onfly=8 AND 
			counter_calls_up_stored=8 AND counter_calls_down_stored<8 THEN
//in prova		
			array_dest_up_onfly_FB[0]:=array_dest_down_stored_FB[0];
			FOR cont := 1 TO 7 BY 1 DO
				array_dest_down_onfly_FB[cont]:=array_dest_down_stored_FB[cont];					
				array_dest_down_stored_FB[cont]:=-1;
			END_FOR;
			sliding_index_3:=sliding_index_4-1;
			sliding_index_4:=0;
			sliding_index_1:=1;
			enable_target_up_down_FB:=TRUE;
		END_IF
	ELSE
		enable_target_up_down_FB:=FALSE;		
	END_IF
	can_be_clicked:=TRUE;
END_IF
target_down_FB:=array_dest_down_onfly_FB[0];
target_up_FB:=array_dest_up_onfly_FB[0];

already_pres:=FALSE; //devo resettarlo ad ogni chiamata per pulire  il flag

counter_calls_up_stored:=0;
counter_calls_down_stored:=0;
counter_calls_up_onfly:=0;
counter_calls_down_onfly:=0;
END_ACTION

ACTION Init_active:
//INIZIALIZZAZIONE DEGLI OUTPUT DI CARDINAL
target_up_FB:=8;
target_down_FB:=-1;
Destination_FB:=0;
enable_target_up_down_FB:=TRUE;

(*Visualization: internal panel variables used to turn on the LED*)
PGVis_FB:=FALSE;
P1Vis_FB:=FALSE;
P2Vis_FB:=FALSE;
P3Vis_FB:=FALSE;
P4Vis_FB:=FALSE;
P5Vis_FB:=FALSE;
P6Vis_FB:=FALSE;
P7Vis_FB:=FALSE;

(*Visualization: external panel variables used to turn on the LED*)
UpDeckGVis_FB:=FALSE;
UpDeck1Vis_FB:=FALSE;
UpDeck2Vis_FB:=FALSE;
UpDeck3Vis_FB:=FALSE;
UpDeck4Vis_FB:=FALSE;
UpDeck5Vis_FB:=FALSE;
UpDeck6Vis_FB:=FALSE;
DownDeck7Vis_FB:=FALSE;
DownDeck6Vis_FB:=FALSE;
DownDeck5Vis_FB:=FALSE;
DownDeck4Vis_FB:=FALSE;
DownDeck3Vis_FB:=FALSE;
DownDeck2Vis_FB:=FALSE;
DownDeck1Vis_FB:=FALSE;

//INIZIALIZZAZIONE ARRAYS AD UN VALORE DI PRIO NON POSSIBILE, OVVERO 8, CON DEST IMPOSSIBILE, SEMPRE 8
FOR sliding_index_1 := 0 TO 7 BY 1 DO
	array_dest_up_onfly_FB[sliding_index_1]:=8;
	array_dest_up_stored_FB[sliding_index_1]:=8;
	
	array_dest_down_onfly_FB[sliding_index_1]:=-1;
	array_dest_down_stored_FB[sliding_index_1]:=-1;
END_FOR;

//INZIALIZZAZIONE INDICI DI SCORRIMENTO ARRAYS


//INIZIALIZZAZIONE DELLE VARIABILI LOCALI 
Dest_floor:=8; //contiene variabile destinazione
can_be_clicked:=TRUE; //permette un'altra chiamata solo dopo aver riordinato l'array
up_motion:=false; //fornisce un verso alle chiamate
cancel_time:=TRUE;
 //indici di utilità per array
k:=0;
k_1:=0;
i:=0;
i_1:=0;
min_index:=8;
min_index_1:=8;
max_index:=8;
max_index_1:=8;
//variabili d'appoggio per riordino
var1:=0;
var1_1:=0;
//indici di scorrimento array per visualizzazione destinazione
sliding_index_1:=0;
sliding_index_2:=0;
sliding_index_3:=0;
sliding_index_4:=0;
//flag di utilità
already_pres:=FALSE;
counter_calls_up_stored:=0;
counter_calls_down_stored:=0;
counter_calls_up_onfly:=0;
counter_calls_down_onfly:=0;
END_ACTION

ACTION Cancel_call_active:
//SE MOVES_MODULE HA ESEGUITO LA CHIAMATA MANDA UN FLAG DI CORRETTO SERVIZIO DI CHIAMATA UP
IF served_up_FB THEN
//DEVO SPEGNERE L'ILLUMINAZIONE DEL TASTO
	IF target_up_FB=0 THEN
		IF PGVis_FB THEN
			PGVis_FB:= FALSE;
		END_IF
		IF UpDeckGVis_FB THEN
			UpDeckGVis_FB:= FALSE;
		END_IF
	END_IF
	IF target_up_FB=1 THEN
		IF P1Vis_FB THEN
			P1Vis_FB:= FALSE;
		END_IF
		IF UpDeck1Vis_FB THEN
			UpDeck1Vis_FB:= FALSE;
		END_IF
		IF DownDeck1Vis_FB THEN
			DownDeck1Vis_FB:= FALSE;
		END_IF
	END_IF
	IF target_up_FB=2 THEN
		IF P2Vis_FB THEN
			P2Vis_FB:= FALSE;
		END_IF
		IF UpDeck2Vis_FB THEN
			UpDeck2Vis_FB:= FALSE;
		END_IF
		IF DownDeck2Vis_FB THEN
			DownDeck2Vis_FB:= FALSE;
		END_IF
	END_IF
	IF target_up_FB=3 THEN
		IF P3Vis_FB THEN
			P3Vis_FB:= FALSE;
		END_IF
		IF UpDeck3Vis_FB THEN
			UpDeck3Vis_FB:= FALSE;
		END_IF
		IF DownDeck3Vis_FB THEN
			DownDeck3Vis_FB:= FALSE;
		END_IF
	END_IF
	IF target_up_FB=4 THEN
		IF P4Vis_FB THEN
			P4Vis_FB:= FALSE;
		END_IF
		IF UpDeck4Vis_FB THEN
			UpDeck4Vis_FB:= FALSE;
		END_IF
		IF DownDeck4Vis_FB THEN
			DownDeck4Vis_FB:= FALSE;
		END_IF
	END_IF
	IF target_up_FB=5 THEN
		IF P5Vis_FB THEN
			P5Vis_FB:= FALSE;
		END_IF
		IF UpDeck5Vis_FB THEN
			UpDeck5Vis_FB:= FALSE;
		END_IF
		IF DownDeck5Vis_FB THEN
			DownDeck5Vis_FB:= FALSE;
		END_IF
	END_IF
	IF target_up_FB=6 THEN
		IF P6Vis_FB THEN
			P6Vis_FB:= FALSE;
		END_IF
		IF UpDeck6Vis_FB THEN
			UpDeck6Vis_FB:= FALSE;
		END_IF
		IF DownDeck6Vis_FB THEN
			DownDeck6Vis_FB:= FALSE;
		END_IF
	END_IF
	IF target_up_FB=7 THEN
		IF P7Vis_FB THEN
			P7Vis_FB:= FALSE;
		END_IF
		IF DownDeck7Vis_FB THEN
			DownDeck7Vis_FB:= FALSE;
		END_IF
	END_IF
//CANCELLO LA CHIAMATA SERVITA DANDOGLI IL VALORE DI PRIO E DEST NON ESISTENTI, OVVERO 8
	array_dest_up_onfly_FB[0]:= 8;
	// array ordinato, qui potrei aggiungere la possibilità di versare stored in onfly
	
// 	IF target_up_FB=8 THEN
// //CONTROLLO IL PRIMO VALORE DELL'ARRAY UP, SE=8 PROVO A VEDERE GLI ALTRI ARRAY	
// 		FOR cont := 0 TO 7 BY 1 DO
// 			IF array_dest_up_onfly_FB[cont]=8 THEN
// 				counter_calls_up_onfly:= counter_calls_up_onfly+1;
// 			END_IF
// 			IF array_dest_down_onfly_FB[cont]=8 THEN
// 				counter_calls_down_onfly:= counter_calls_down_onfly+1;
// 			END_IF
// 			IF array_dest_up_stored_FB[cont]=8 THEN
// 				counter_calls_up_stored:= counter_calls_up_stored+1;
// 			END_IF
// 			IF array_dest_down_stored_FB[cont]=-1 THEN
// 				counter_calls_down_stored:= counter_calls_down_stored+1;
// 			END_IF
// 		END_FOR
// //ORA PROCEDO ALLE CASISTICHE
// (*CASO CON:
// FLY_UP VUOTO
// FLY_DOWN PIENO
// STORED_UP INDIFFERENTE
// STORED_DOWN INDIFFERENTE
// COPIO LE CHIAMATE STORED_UP IN FLY_UP MENTRE SERVO FLY_DOWN
//  *)
// 		IF 	counter_calls_up_onfly=8 AND counter_calls_down_onfly<8 AND 
// 			counter_calls_up_stored<=8 AND counter_calls_down_stored<=8 THEN	
// 
// 			FOR cont := 0 TO 7 BY 1 DO
// 				array_dest_up_onfly_FB[cont]:=array_dest_up_stored_FB[cont];
// 				array_prio_up_onfly_FB[cont]:=array_prio_up_stored_FB[cont];
// 				array_dest_up_stored_FB[cont]:=8;
// 				array_prio_up_stored_FB[cont]:=8;
// 			END_FOR;
// 			sliding_index_1:=sliding_index_2;
// 			sliding_index_2:=0;
// 		END_IF
// (*CASO CON:
// FLY_UP VUOTO
// FLY_DOWN VUOTO
// STORED_UP PIENO
// STORED_DOWN VUOTO
// COPIO LA PRIMA CALL IN FLY_DOWN E LE ALTRE IN FLY_UP, IN MODO CHE POSSA TORNARE GIù FINO ALLA 
// CALL CON DESTINAZIONE MINORE
// *)
// //CASO CON STORED_DOWN VUOTO E STORED_UP PIENO, COPIO LE CHIAMATE STORED_UP IN FLY_DOWN	
// 		IF 	counter_calls_up_onfly=8 AND counter_calls_down_onfly=8 AND 
// 			counter_calls_up_stored<8 AND counter_calls_down_stored=8 THEN
// //in prova		
// 			array_dest_down_onfly_FB[0]:=array_dest_up_stored_FB[0];
// 			array_prio_down_onfly_FB[0]:=array_prio_up_stored_FB[0];
// 			FOR cont := 1 TO 7 BY 1 DO
// 				array_dest_up_onfly_FB[cont]:=array_dest_up_stored_FB[cont];
// 				array_prio_up_onfly_FB[cont]:=array_prio_up_stored_FB[cont];
// 				array_dest_up_stored_FB[cont]:=8;
// 				array_prio_up_stored_FB[cont]:=8;
// 			END_FOR;
// 			sliding_index_1:=sliding_index_2-1;
// 			sliding_index_2:=0;
// 			sliding_index_3:=1;
// // 			enable_target_up_down_FB:=FALSE;
// 		END_IF
// 	counter_calls_up_stored:=0;
// 	counter_calls_down_stored:=0;
// 	counter_calls_up_onfly:=0;
// 	counter_calls_down_onfly:=0;
// 	END_IF
END_IF

//RIORDINO L'ARRAY UP
k_1:=0;	
i_1:=0;	
WHILE i_1<=7 DO
	k_1:=i_1+1;
	min_index_1:=i_1;
	WHILE k_1<=7 DO
		IF array_dest_up_onfly_FB[k_1]<array_dest_up_onfly_FB[i_1] THEN
			min_index_1:=k_1;
		END_IF	
		k_1:=k_1+1;
	END_WHILE
	var1_1:= array_dest_up_onfly_FB[i_1];
	array_dest_up_onfly_FB[i_1]:=array_dest_up_onfly_FB[min_index_1];
	array_dest_up_onfly_FB[min_index_1]:=var1_1;
	i_1:=i_1+1;
END_WHILE
target_up_FB:=array_dest_up_onfly_FB[0];

//SE MOVES_MODULE HA ESEGUITO LA CHIAMATA MANDA UN FLAG DI CORRETTO SERVIZIO DI CHIAMATA DOWN

IF served_down_FB THEN
//DEVO ANCHE SPEGNERE L'ILLUMINAZIONE DEL TASTO
	IF target_down_FB=0 THEN
		IF PGVis_FB THEN
			PGVis_FB:= FALSE;
		END_IF
		IF UpDeckGVis_FB THEN
			UpDeckGVis_FB:= FALSE;
		END_IF
	END_IF
	IF target_down_FB=1 THEN
		IF P1Vis_FB THEN
			P1Vis_FB:= FALSE;
		END_IF
		IF UpDeck1Vis_FB THEN
			UpDeck1Vis_FB:= FALSE;
		END_IF
		IF DownDeck1Vis_FB THEN
			DownDeck1Vis_FB:= FALSE;
		END_IF
	END_IF
	IF target_down_FB=2 THEN
		IF P2Vis_FB THEN
			P2Vis_FB:= FALSE;
		END_IF
		IF UpDeck2Vis_FB THEN
			UpDeck2Vis_FB:= FALSE;
		END_IF
		IF DownDeck2Vis_FB THEN
			DownDeck2Vis_FB:= FALSE;
		END_IF
	END_IF
	IF target_down_FB=3 THEN
		IF P3Vis_FB THEN
			P3Vis_FB:= FALSE;
		END_IF
		IF UpDeck3Vis_FB THEN
			UpDeck3Vis_FB:= FALSE;
		END_IF
		IF DownDeck3Vis_FB THEN
			DownDeck3Vis_FB:= FALSE;
		END_IF
	END_IF
	IF target_down_FB=4 THEN
		IF P4Vis_FB THEN
			P4Vis_FB:= FALSE;
		END_IF
		IF UpDeck4Vis_FB THEN
			UpDeck4Vis_FB:= FALSE;
		END_IF
		IF DownDeck4Vis_FB THEN
			DownDeck4Vis_FB:= FALSE;
		END_IF
	END_IF
	IF target_down_FB=5 THEN
		IF P5Vis_FB THEN
			P5Vis_FB:= FALSE;
		END_IF
		IF UpDeck5Vis_FB THEN
			UpDeck5Vis_FB:= FALSE;
		END_IF
		IF DownDeck5Vis_FB THEN
			DownDeck5Vis_FB:= FALSE;
		END_IF
	END_IF
	IF target_down_FB=6 THEN
		IF P6Vis_FB THEN
			P6Vis_FB:= FALSE;
		END_IF
		IF UpDeck6Vis_FB THEN
			UpDeck6Vis_FB:= FALSE;
		END_IF
		IF DownDeck6Vis_FB THEN
			DownDeck6Vis_FB:= FALSE;
		END_IF
	END_IF
	IF target_down_FB=7 THEN
		IF P7Vis_FB THEN
			P7Vis_FB:= FALSE;
		END_IF
		IF DownDeck7Vis_FB THEN
			DownDeck7Vis_FB:= FALSE;
		END_IF
	END_IF
	array_dest_down_onfly_FB[0]:= -1;
	// array ordinato, qui potrei aggiungere la possibilità di versare stored in onfly
	
// 	IF target_down_FB=8 THEN
// //CONTROLLO IL PRIMO VALORE DELL'ARRAY UP, SE=8 PROVO A VEDERE GLI ALTRI ARRAY	
// 		FOR cont := 0 TO 7 BY 1 DO
// 			IF array_dest_up_onfly_FB[cont]=8 THEN
// 				counter_calls_up_onfly:= counter_calls_up_onfly+1;
// 			END_IF
// 			IF array_dest_down_onfly_FB[cont]=8 THEN
// 				counter_calls_down_onfly:= counter_calls_down_onfly+1;
// 			END_IF
// 			IF array_dest_up_stored_FB[cont]=8 THEN
// 				counter_calls_up_stored:= counter_calls_up_stored+1;
// 			END_IF
// 			IF array_dest_down_stored_FB[cont]=-1 THEN
// 				counter_calls_down_stored:= counter_calls_down_stored+1;
// 			END_IF
// 		END_FOR
// //ORA PROCEDO ALLE CASISTICHE
// (*CASO CON:
// FLY_UP PIENO
// FLY_DOWN VUOTO
// STORED_UP INDIFFERENTE
// STORED_DOWN INDIFFERENTE
// COPIO LE CHIAMATE STORED_DOWN IN FLY_DOWN MENTRE SERVO FLY_UP
//  *)
// 		IF 	counter_calls_up_onfly<8 AND counter_calls_down_onfly=8 AND 
// 			counter_calls_up_stored<=8 AND counter_calls_down_stored<=8 THEN	
// 
// 			FOR cont := 0 TO 7 BY 1 DO
// 				IF array_dest_down_stored_FB[cont]=-1 THEN
// 					array_dest_down_onfly_FB[cont]:=8;
// 				ELSE
// 					array_dest_down_onfly_FB[cont]:=array_dest_down_stored_FB[cont];					
// 				END_IF
// 				array_prio_down_onfly_FB[cont]:=array_prio_down_stored_FB[cont];
// 				array_dest_down_stored_FB[cont]:=-1;
// 				array_prio_down_stored_FB[cont]:=8;
// 			END_FOR;
// 			sliding_index_3:=sliding_index_4;
// 			sliding_index_4:=0;
// // 			enable_target_up_down_FB:=TRUE;
// 		END_IF
// (*CASO CON:
// FLY_UP VUOTO
// FLY_DOWN VUOTO
// STORED_UP VUOTO
// STORED_DOWN PIENO
// COPIO LA PRIMA CALL IN FLY_UP E LE ALTRE IN FLY_DOWN, IN MODO CHE POSSA TORNARE SU FINO ALLA 
// CALL CON DESTINAZIONE MAGGIORE
// *)
// 		IF 	counter_calls_up_onfly=8 AND counter_calls_down_onfly=8 AND 
// 			counter_calls_up_stored=8 AND counter_calls_down_stored<8 THEN
// //in prova		
// 			array_dest_up_onfly_FB[0]:=array_dest_down_stored_FB[0];
// 			array_prio_up_onfly_FB[0]:=array_prio_down_stored_FB[0];
// 			FOR cont := 1 TO 7 BY 1 DO
// 				IF array_dest_down_stored_FB[cont]=-1 THEN
// 					array_dest_down_onfly_FB[cont]:=8;
// 				ELSE
// 					array_dest_down_onfly_FB[cont]:=array_dest_down_stored_FB[cont];					
// 				END_IF
// 				array_prio_down_onfly_FB[cont]:=array_prio_down_stored_FB[cont];
// 				array_dest_down_stored_FB[cont]:=-1;
// 				array_prio_down_stored_FB[cont]:=8;
// 			END_FOR;
// 			sliding_index_3:=sliding_index_4-1;
// 			sliding_index_4:=0;
// 			sliding_index_1:=1;
// // 			enable_target_up_down_FB:=TRUE;
// 		END_IF
// 	counter_calls_up_stored:=0;
// 	counter_calls_down_stored:=0;
// 	counter_calls_up_onfly:=0;
// 	counter_calls_down_onfly:=0;			
// 	END_IF

END_IF
//RIORDINO L'ARRAY DOWN
k_1:=0;
i_1:=0;
WHILE i_1<=7 DO
	k_1:=i_1+1;
	max_index_1:=i_1;
	WHILE k_1<=7 DO
		IF array_dest_down_onfly_FB[k_1]>array_dest_down_onfly_FB[i_1] THEN
			max_index_1:=k_1;
		END_IF	
		k_1:=k_1+1;
		END_WHILE
	var1_1:= array_dest_down_onfly_FB[i_1];
	array_dest_down_onfly_FB[i_1]:=array_dest_down_onfly_FB[max_index_1];
	array_dest_down_onfly_FB[max_index_1]:=var1_1;		
	i_1:=i_1+1;
END_WHILE
target_down_FB:=array_dest_down_onfly_FB[0];

//AGGIORNAMENTO TARGET
IF Up_FB THEN
	Destination_FB:= target_up_FB;
ELSE
	Destination_FB:= target_down_FB;
END_IF
END_ACTION

END_FUNCTION_BLOCK

// Device/Application/GAs/Moves_module
FUNCTION_BLOCK Moves_module
VAR_INPUT	
	Start_: BOOL;
	StartWhat: STRING;
	Stop: BOOL;
	
//INPUT PROVENIENTI DA CARDINAL
	target_up_FB: INT; //valore da dare a Dest_target_up
	target_down_FB: INT; //valore da dare a Dest_target_down
	enable_target_up_down_FB: BOOL;
	
// SENSORI
	DeckSensor_FB: BOOL;
	RampSensor_FB: BOOL;
	LimitDown_FB: BOOL;
	LimitUp_FB: BOOL;
	
	Emergency_FB: BOOL;
END_VAR
VAR_OUTPUT
	State: STRING;
	Done: BOOL;	
//OUTPUT VERSO CARDINAL
	served_up_FB: BOOL; //flag di finito servizio del valore target_up
	served_down_FB: BOOL; //flag di finito servizio del valore target_down
//OUTPUT VERSO LA POLICY
	Current_FB: INT; //variabile di visualizzazione piano corrente
	Up_FB: BOOL; //manovra il verso dell'ascensore
	Motor_on_FB: BOOL; //accende o spegne il motore dell'ascensore
	Vel_FB: BOOL; //manovra la velocità dell'ascensore
	deck_error_FB: BOOL; //flag per gestire errore di deck
	ramp_error_FB: BOOL; //flag per gestire errore di ramp	
	EmergencyVis_FB: BOOL;
	
	G_floor_prob: BOOL;
END_VAR
VAR
	sync: BOOL;
	Opok: BOOL;
	ramp_counter: INT;
	deck_counter: INT;
END_VAR

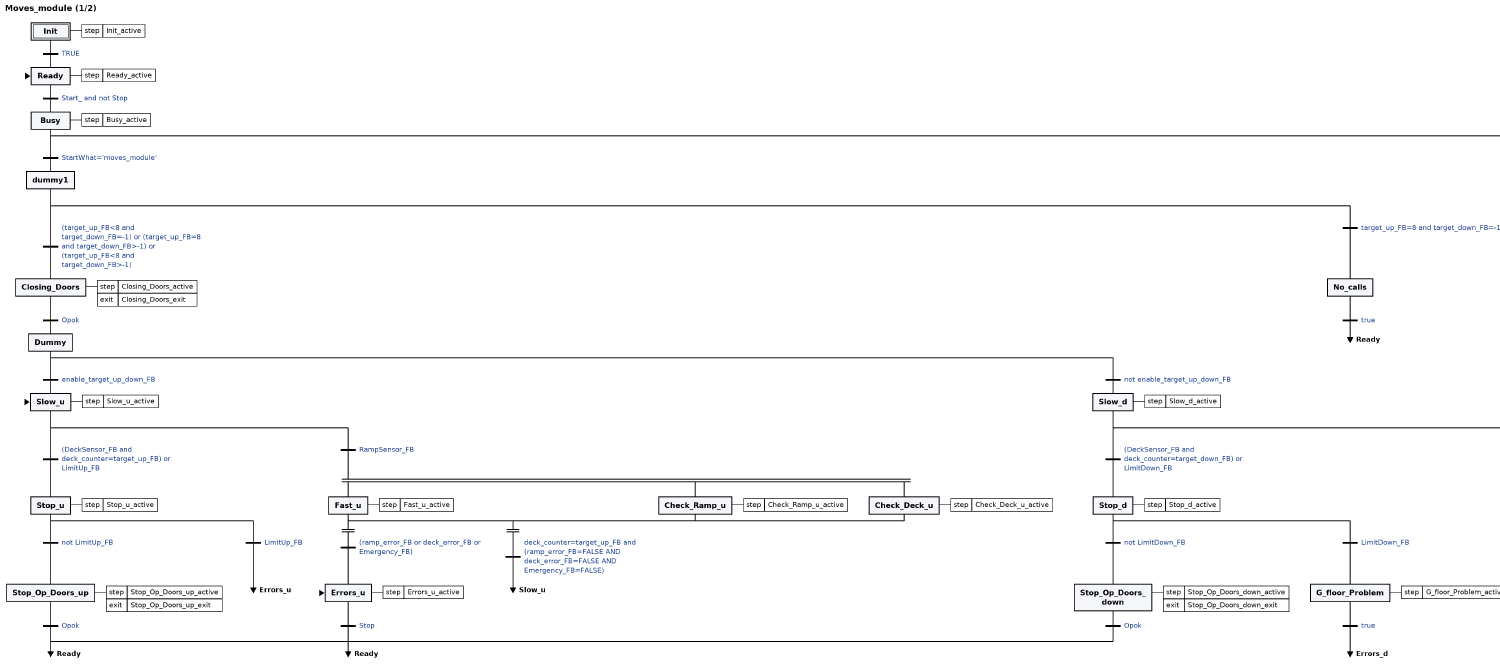
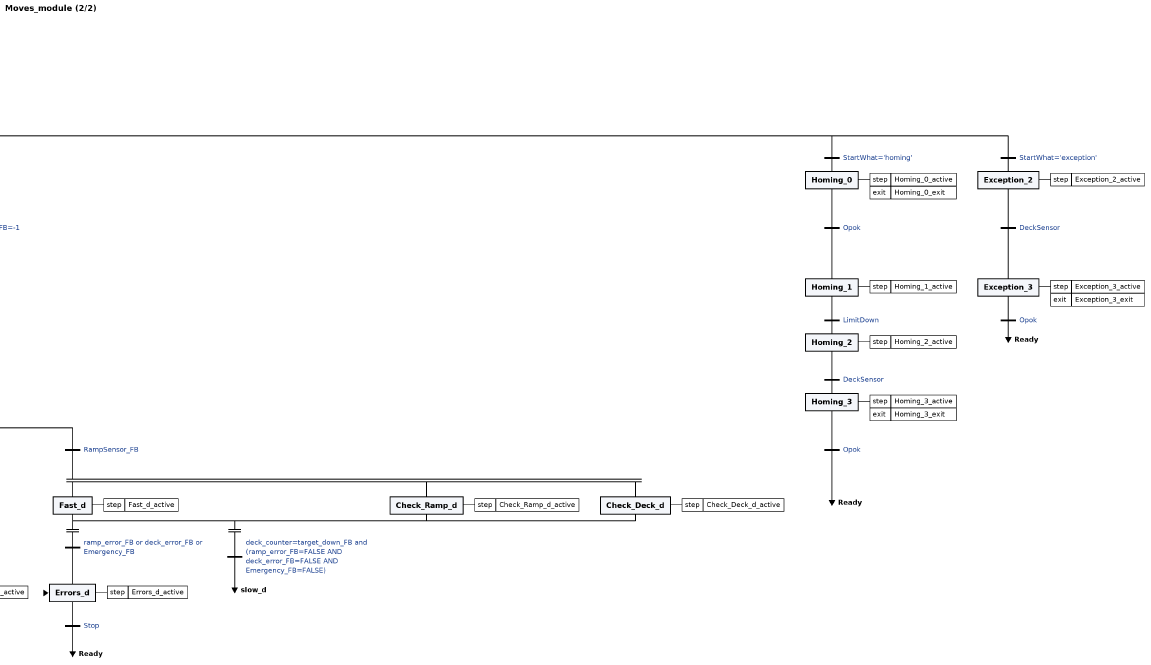
INITIAL_STEP Init:
    Init_active(N);  // step action
END_STEP
TRANSITION FROM Init TO Ready
    := TRUE;
END_TRANSITION
STEP Ready:
    Ready_active(N);  // step action
END_STEP
TRANSITION FROM Ready TO Busy
    := Start_ and not Stop;
END_TRANSITION
STEP Busy:
    Busy_active(N);  // step action
END_STEP
TRANSITION FROM Busy TO dummy1
    := StartWhat='moves_module';
END_TRANSITION
STEP dummy1:
END_STEP
TRANSITION FROM Busy TO Homing_0
    := StartWhat='homing';
END_TRANSITION
STEP Homing_0:
    Homing_0_active(N);  // step action
    Homing_0_exit(P0);  // exit action
END_STEP
TRANSITION FROM Homing_0 TO Homing_1
    := Opok;
END_TRANSITION
STEP Homing_1:
    Homing_1_active(N);  // step action
END_STEP
TRANSITION FROM Homing_1 TO Homing_2
    := LimitDown;
END_TRANSITION
STEP Homing_2:
    Homing_2_active(N);  // step action
END_STEP
TRANSITION FROM Homing_2 TO Homing_3
    := DeckSensor;
END_TRANSITION
STEP Homing_3:
    Homing_3_active(N);  // step action
    Homing_3_exit(P0);  // exit action
END_STEP
TRANSITION FROM Homing_3 TO Ready
    := Opok;
END_TRANSITION
TRANSITION FROM Busy TO Exception_2
    := StartWhat='exception';
END_TRANSITION
STEP Exception_2:
    Exception_2_active(N);  // step action
END_STEP
TRANSITION FROM Exception_2 TO Exception_3
    := DeckSensor;
END_TRANSITION
STEP Exception_3:
    Exception_3_active(N);  // step action
    Exception_3_exit(P0);  // exit action
END_STEP
TRANSITION FROM Exception_3 TO Ready
    := Opok;
END_TRANSITION
TRANSITION FROM dummy1 TO Closing_Doors
    := (target_up_FB<8 and target_down_FB=-1) or (target_up_FB=8 and target_down_FB>-1) or (target_up_FB<8 and target_down_FB>-1);
END_TRANSITION
STEP Closing_Doors:
    Closing_Doors_active(N);  // step action
    Closing_Doors_exit(P0);  // exit action
END_STEP
TRANSITION FROM Closing_Doors TO Dummy
    := Opok;
END_TRANSITION
STEP Dummy:
END_STEP
TRANSITION FROM Dummy TO Slow_u
    := enable_target_up_down_FB;
END_TRANSITION
STEP Slow_u:
    Slow_u_active(N);  // step action
END_STEP
TRANSITION FROM Slow_u TO Stop_u
    := (DeckSensor_FB and deck_counter=target_up_FB) or LimitUp_FB;
END_TRANSITION
STEP Stop_u:
    Stop_u_active(N);  // step action
END_STEP
TRANSITION FROM Stop_u TO Stop_Op_Doors_up
    := not LimitUp_FB;
END_TRANSITION
TRANSITION FROM Stop_u TO Errors_u
    := LimitUp_FB;
END_TRANSITION
STEP Stop_Op_Doors_up:
    Stop_Op_Doors_up_active(N);  // step action
    Stop_Op_Doors_up_exit(P0);  // exit action
END_STEP
TRANSITION FROM Stop_Op_Doors_up TO Ready
    := Opok;
END_TRANSITION
TRANSITION FROM Slow_u TO (Fast_u, Check_Ramp_u, Check_Deck_u)
    := RampSensor_FB;
END_TRANSITION
STEP Fast_u:
    Fast_u_active(N);  // step action
END_STEP
STEP Check_Ramp_u:
    Check_Ramp_u_active(N);  // step action
END_STEP
STEP Check_Deck_u:
    Check_Deck_u_active(N);  // step action
END_STEP
TRANSITION FROM (Fast_u, Check_Ramp_u, Check_Deck_u) TO Errors_u
    := (ramp_error_FB or deck_error_FB or Emergency_FB);
END_TRANSITION
STEP Errors_u:
    Errors_u_active(N);  // step action
END_STEP
TRANSITION FROM Errors_u TO Ready
    := Stop;
END_TRANSITION
TRANSITION FROM (Fast_u, Check_Ramp_u, Check_Deck_u) TO Slow_u
    := deck_counter=target_up_FB and (ramp_error_FB=FALSE AND deck_error_FB=FALSE AND Emergency_FB=FALSE);
END_TRANSITION
TRANSITION FROM Dummy TO Slow_d
    := not enable_target_up_down_FB;
END_TRANSITION
STEP Slow_d:
    Slow_d_active(N);  // step action
END_STEP
TRANSITION FROM Slow_d TO Stop_d
    := (DeckSensor_FB and deck_counter=target_down_FB) or LimitDown_FB;
END_TRANSITION
STEP Stop_d:
    Stop_d_active(N);  // step action
END_STEP
TRANSITION FROM Stop_d TO Stop_Op_Doors_down
    := not LimitDown_FB;
END_TRANSITION
TRANSITION FROM Stop_d TO G_floor_Problem
    := LimitDown_FB;
END_TRANSITION
STEP G_floor_Problem:
    G_floor_Problem_active(N);  // step action
END_STEP
TRANSITION FROM G_floor_Problem TO Errors_d
    := true;
END_TRANSITION
STEP Stop_Op_Doors_down:
    Stop_Op_Doors_down_active(N);  // step action
    Stop_Op_Doors_down_exit(P0);  // exit action
END_STEP
TRANSITION FROM Stop_Op_Doors_down TO Ready
    := Opok;
END_TRANSITION
TRANSITION FROM Slow_d TO (Fast_d, Check_Ramp_d, Check_Deck_d)
    := RampSensor_FB;
END_TRANSITION
STEP Fast_d:
    Fast_d_active(N);  // step action
END_STEP
STEP Check_Ramp_d:
    Check_Ramp_d_active(N);  // step action
END_STEP
STEP Check_Deck_d:
    Check_Deck_d_active(N);  // step action
END_STEP
TRANSITION FROM (Fast_d, Check_Ramp_d, Check_Deck_d) TO Errors_d
    := ramp_error_FB or deck_error_FB or Emergency_FB;
END_TRANSITION
STEP Errors_d:
    Errors_d_active(N);  // step action
END_STEP
TRANSITION FROM Errors_d TO Ready
    := Stop;
END_TRANSITION
TRANSITION FROM (Fast_d, Check_Ramp_d, Check_Deck_d) TO slow_d
    := deck_counter=target_down_FB and (ramp_error_FB=FALSE AND deck_error_FB=FALSE AND Emergency_FB=FALSE);
END_TRANSITION
TRANSITION FROM dummy1 TO No_calls
    := target_up_FB=8 and target_down_FB=-1;
END_TRANSITION
STEP No_calls:
END_STEP
TRANSITION FROM No_calls TO Ready
    := true;
END_TRANSITION

ACTION G_floor_Problem_active:
G_floor_prob:=TRUE;
END_ACTION

ACTION Stop_Op_Doors_down_active:
// RESETTO FLAG DI SERVIZIO CHIAMATA EFFETTUATO
served_down_FB:=FALSE;
//APERTURA PORTE 
IF door_module_0.State='ready' THEN
	door_module_0.Do_:=TRUE;
	door_module_0.DoWhat:='open_door';
END_IF

IF door_module_0.Done AND door_module_0.State='busy' THEN
	door_module_0.Do_:=FALSE;
	sync:=TRUE;
END_IF

Opok:= sync AND NOT door_module_0.Done;
END_ACTION

ACTION Ready_active:
State:='ready'; 
ramp_error_FB:=FALSE; //flag per gestire errore di ramp
deck_error_FB:=FALSE; //flag per gestire errore di deck
Done:=FALSE;
END_ACTION

ACTION Busy_active:
State:='busy';
G_floor_prob:=FALSE;
EmergencyVis_FB:=FALSE;
IF NOT enable_target_up_down_FB OR Current_FB=7 THEN
	Up_FB:=FALSE;
END_IF

IF enable_target_up_down_FB OR Current_FB=0 THEN
	Up_FB:=TRUE;
END_IF
END_ACTION

ACTION Closing_Doors_active:
//CHIUSURA PORTE 
IF door_module_0.State='ready' THEN
	door_module_0.Do_:=TRUE;
	door_module_0.DoWhat:='close_door';
END_IF

IF door_module_0.Done AND door_module_0.State='busy' THEN
	door_module_0.Do_:=FALSE;
	sync:=TRUE;
END_IF

Opok:= sync and not door_module_0.Done;
END_ACTION

ACTION Closing_Doors_exit:
sync:=FALSE;
Opok:=FALSE;
END_ACTION

ACTION Init_active:
//INIZIALIZZAZIONE DELLE VARIABILI OUTPUT DI MOVES_MODULE

//OUTPUT VERSO CARDINAL
served_up_FB:=FALSE; //flag di finito servizio del valore target_up
served_down_FB:=FALSE; //flag di finito servizio del valore target_down

//OUTPUT VERSO LA POLICY
//Current_FB:=8; //variabile di visualizzazione piano corrente
Up_FB:=TRUE; //manovra il verso dell'ascensore, inizializzo true perchè dopo homing può andare solo su
Motor_on_FB:=FALSE; //accende o spegne il motore dell'ascensore
Vel_FB:=FALSE; //manovra la velocità dell'ascensore
// deck_error_FB:=FALSE; //flag per gestire errore di deck
// deck_error_FB:=FALSE; //flag per gestire errore di ramp

//VARIABILI LOCALI DEL FB
sync:=FALSE;
Opok:=FALSE;
ramp_counter:=0;
deck_counter:=0;
END_ACTION

ACTION Stop_Op_Doors_down_exit:
sync:=FALSE;
Opok:=FALSE;
END_ACTION

ACTION Slow_d_active:
ramp_counter:=0;
//DISCESA VERSO IL BASSO
Motor_on_FB:= TRUE;
Up_FB:= FALSE;
Vel_FB:= FALSE;
END_ACTION

ACTION Stop_Op_Doors_up_active:
// RESETTO FLAG DI SERVIZIO CHIAMATA EFFETTUATO
served_up_FB:=FALSE;
//APERTURA PORTE 
IF door_module_0.State='ready' THEN
	door_module_0.Do_:=TRUE;
	door_module_0.DoWhat:='open_door';
END_IF

IF door_module_0.Done AND door_module_0.State='busy' THEN
	door_module_0.Do_:=FALSE;
	sync:=TRUE;

END_IF

Opok:= sync AND NOT door_module_0.Done;
END_ACTION

ACTION Slow_u_active:
ramp_counter:=0;
//SALITA VERSO L'ALTO
Motor_on_FB:= TRUE;
Up_FB:= TRUE;
Vel_FB:= FALSE;
END_ACTION

ACTION Fast_u_active:
//SALITA VERSO L'ALTO
Motor_on_FB:= TRUE;
Up_FB:= TRUE;
Vel_FB:= TRUE;
END_ACTION

ACTION Stop_Op_Doors_up_exit:
sync:=FALSE;
Opok:=FALSE;
END_ACTION

ACTION Check_Ramp_u_active:
//CONTROLLO DEL RAMPSENSOR
IF RampSensor THEN
	ramp_counter:=ramp_counter+1;
	IF ramp_counter=2 THEN
		deck_counter:=deck_counter+1;
	END_IF
	IF ramp_counter=3 THEN
		deck_error_FB:=TRUE;
	END_IF
END_IF
END_ACTION

ACTION Check_Deck_u_active:
//CONTROLLO DEL DECKSENSOR
IF DeckSensor THEN
	IF ramp_counter=1 THEN
		ramp_error_FB:=TRUE;
	END_IF
	ramp_counter:=0;
	IF Current_FB<deck_counter THEN
		Current_FB:=Current_FB+1;	
	END_IF
END_IF
END_ACTION

ACTION Fast_d_active:
//DISCESA VERSO IL BASSO 
Motor_on_FB:= TRUE;
Up_FB:= FALSE;
Vel_FB:= TRUE;

IF LimitDown_FB THEN
	deck_error_FB:=TRUE;
END_IF
END_ACTION

ACTION Check_Ramp_d_active:
//CONTROLLO DEL RAMPSENSOR
IF RampSensor THEN
	ramp_counter:=ramp_counter+1;
	IF ramp_counter=2 THEN
		deck_counter:=deck_counter-1;
	END_IF
	IF ramp_counter=3 THEN
			deck_error_FB:=TRUE;
	END_IF
END_IF
END_ACTION

ACTION Check_Deck_d_active:
//CONTROLLO DEL DECKSENSOR
IF DeckSensor THEN
	IF ramp_counter=1 THEN
		ramp_error_FB:=TRUE;
	END_IF
	ramp_counter:=0;
	IF Current_FB>deck_counter THEN
		Current_FB:=Current_FB-1;	
	END_IF
END_IF
END_ACTION

ACTION Stop_u_active:
IF LimitUp_FB THEN
//STOP
	Motor_on_FB:=FALSE;
	deck_error_FB:=TRUE;
ELSE
//STOP
	Motor_on_FB:=FALSE; 
	Current_FB:=Current_FB+1;
// MANDO FLAG DI SERVIZIO CHIAMATA EFFETTUATO
	served_up_FB:=TRUE;
END_IF
END_ACTION

ACTION Stop_d_active:
IF LimitDown_FB THEN
//STOP
	Motor_on_FB:=FALSE;
	deck_error_FB:=TRUE;
ELSE
//STOP
	Motor_on_FB:=FALSE;
	Current_FB:=Current_FB-1;
// MANDO FLAG DI SERVIZIO CHIAMATA EFFETTUATO
	served_down_FB:=TRUE;
END_IF
END_ACTION

ACTION Errors_d_active:
//STOP AI MOVIMENTI
Motor_on_FB:=FALSE;
//SE VIENE CHIAMATA EMERGENZA DEVO ACCENDERE IL LED DI EMERGENZA
IF Emergency_FB THEN
	EmergencyVis_FB:=TRUE;
END_IF
IF NOT G_floor_prob THEN
	Current_FB:=0;
ELSE
deck_counter:=1;		
END_IF
END_ACTION

ACTION Errors_u_active:
//STOP AI MOVIMENTI
Motor_on_FB:=FALSE;
// SE VIENE CHIAMATA EMERGENZA DEVO ACCENDERE IL LED DI EMERGENZA
IF Emergency_FB THEN
	EmergencyVis_FB:=TRUE;
END_IF
deck_counter:=0;
Current_FB:=0;
END_ACTION

ACTION Homing_0_active:
//APERTURA PORTE 
IF door_module_0.State='ready' THEN
	door_module_0.Do_:=TRUE;
	door_module_0.DoWhat:='close_door';
END_IF

IF door_module_0.Done AND door_module_0.State='busy' THEN
	door_module_0.Do_:=FALSE;
	sync:=TRUE;
END_IF

Opok:= sync and not door_module_0.Done;
END_ACTION

ACTION Homing_0_exit:
sync:=FALSE;
Opok:=FALSE;
END_ACTION

ACTION Homing_1_active:
//HOMING
Motor_on_FB:= TRUE;
Up_FB:= FALSE;
Vel_FB:= FALSE;
END_ACTION

ACTION Homing_2_active:
//HOMING_1
Motor_on_FB:= TRUE;
Up_FB:= TRUE;
Vel_FB:= FALSE;
END_ACTION

ACTION Homing_3_active:
//STOP
Motor_on_FB:= FALSE;
Current_FB:=0;
//APERTURA PORTE 
IF door_module_0.State='ready' THEN
	door_module_0.Do_:=TRUE;
	door_module_0.DoWhat:='open_door';
END_IF

IF door_module_0.Done AND door_module_0.State='busy' THEN
	door_module_0.Do_:=FALSE;
	sync:=TRUE;
	Moves_module_0.Done:=TRUE;
	//SE SI E' MANIFESTATO UN RICHIAMO DI EMERGENCY
	IF EmergencyVis_FB THEN
		Emergency_FB:=FALSE;
	END_IF
END_IF
Opok:= sync AND NOT door_module_0.Done;
END_ACTION

ACTION Homing_3_exit:
sync:=FALSE;
Opok:=FALSE;
END_ACTION

ACTION Exception_2_active:
//VERSO L'ALTO
Motor_on_FB:= TRUE;
Up_FB:= TRUE;
Vel_FB:= FALSE;
END_ACTION

ACTION Exception_3_active:
//STOP
Motor_on_FB:= FALSE;
//SE SI E' MANIFESTATA UN PROBLEMA AL PIANO ZERO (PARTICOLARITA')
Current_FB:=1;
//APERTURA PORTE 
IF door_module_0.State='ready' THEN
	door_module_0.Do_:=TRUE;
	door_module_0.DoWhat:='open_door';
END_IF

IF door_module_0.Done AND door_module_0.State='busy' THEN
	door_module_0.Do_:=FALSE;
	sync:=TRUE;
	Moves_module_0.Done:=TRUE;
	//SE SI E' MANIFESTATO UN RICHIAMO DI EMERGENCY
	IF EmergencyVis_FB THEN
		Emergency_FB:=FALSE;
	END_IF
END_IF
Opok:= sync AND NOT door_module_0.Done;
END_ACTION

ACTION Exception_3_exit:
sync:=FALSE;
Opok:=FALSE;
END_ACTION

END_FUNCTION_BLOCK

// Device/Application/Policy
PROGRAM Policy
VAR
	sync: BOOL;
	Opok: BOOL;
END_VAR

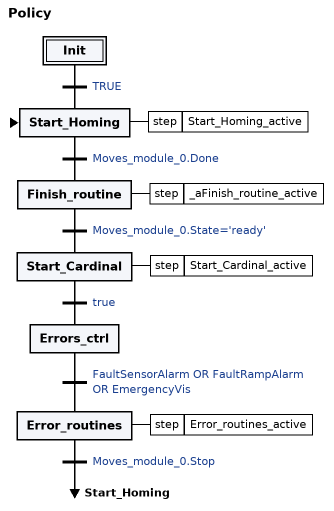
INITIAL_STEP Init:
END_STEP
TRANSITION FROM Init TO Start_Homing
    := TRUE;
END_TRANSITION
STEP Start_Homing:
    Start_Homing_active(N);  // step action
END_STEP
TRANSITION FROM Start_Homing TO Finish_routine
    := Moves_module_0.Done;
END_TRANSITION
STEP Finish_routine:
    _aFinish_routine_active(N);  // step action
END_STEP
TRANSITION FROM Finish_routine TO Start_Cardinal
    := Moves_module_0.State='ready';
END_TRANSITION
STEP Start_Cardinal:
    Start_Cardinal_active(N);  // step action
END_STEP
TRANSITION FROM Start_Cardinal TO Errors_ctrl
    := true;
END_TRANSITION
STEP Errors_ctrl:
END_STEP
TRANSITION FROM Errors_ctrl TO Error_routines
    := FaultSensorAlarm OR FaultRampAlarm OR EmergencyVis;
END_TRANSITION
STEP Error_routines:
    Error_routines_active(N);  // step action
END_STEP
TRANSITION FROM Error_routines TO Start_Homing
    := Moves_module_0.Stop;
END_TRANSITION

ACTION Start_Cardinal_active:
//START DI CARDINAL
IF Cardinal_0.State='ready' THEN
	Cardinal_0.Start_:=TRUE;
	Cardinal_0.Stop:=FALSE;
END_IF
//START DI MOVES_MODULE
IF Moves_module_0.State='ready' THEN
	Moves_module_0.Start_:=TRUE;
	Moves_module_0.Stop:=FALSE;
	Moves_module_0.StartWhat:='moves_module';
END_IF
END_ACTION

ACTION Error_routines_active:
// //STOP DI CARDINAL
// IF Cardinal_0.State='busy' THEN
// 	Cardinal_0.Start_:=FALSE;
// 	Cardinal_0.Stop:=TRUE;
// END_IF
//STOP DI MOVES_MODULE
IF Moves_module_0.State='busy' THEN
	Moves_module_0.Start_:=FALSE;
	Moves_module_0.Stop:=TRUE;
END_IF
END_ACTION

ACTION Start_Homing_active:
//CONTROLLO INIZIALE SULL'HOMING
IF NOT G_floor_problem THEN
	// START DELLA ROUTINE DI HOMING
	IF Moves_module_0.State='ready' THEN
		Moves_module_0.Start_:=TRUE;
		Moves_module_0.Stop:=FALSE;
		Moves_module_0.StartWhat:='homing';
	END_IF
ELSE
	// START DELLA ROUTINE DI EXCEPTION
	IF Moves_module_0.State='ready' THEN
		Moves_module_0.Start_:=TRUE;
		Moves_module_0.Stop:=FALSE;
		Moves_module_0.StartWhat:='exception';
	END_IF
END_IF
END_ACTION

ACTION Start_What_active:




















//START DI MOVES_MODULE
IF Moves_module_0.State='ready' THEN
	Moves_module_0.Start_:=TRUE;
	Moves_module_0.Stop:=FALSE;
END_IF

//STOP DI MOVES_MODULE
IF Moves_module_0.State='busy' THEN
	Moves_module_0.Start_:=FALSE;
	Moves_module_0.Stop:=TRUE;
END_IF
END_ACTION

ACTION _aFinish_routine_active:
// STOP DELLA ROUTINE STARTWHAT
IF Moves_module_0.State='busy' AND Moves_module_0.Done THEN
	Moves_module_0.Start_:=FALSE;
	Moves_module_0.Stop:=TRUE;
END_IF
END_ACTION

END_PROGRAM

// Device/Application/Visualization
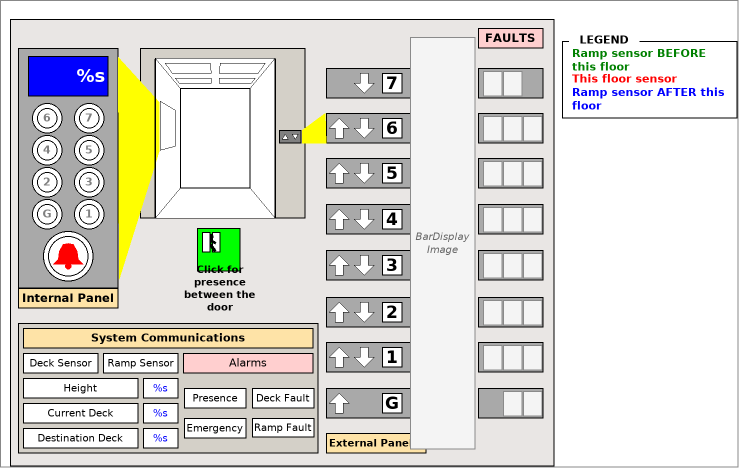
VISUALIZATION Visualization  // 739x468
    Rectangle (10,19 544x447)
    Rectangle (197,228 43x43), colour toggle: GVL.Presence
    Rectangle (18,323 300x130)
    Rectangle (326,433 100x20), "External Panels"
    Rectangle (326,342 100x30)
    Rectangle (382,347 20x20), "1"
    Polygon (354,357) (360,357) (360,347) (368,347) (368,357) (374,357) (364,367), colour toggle: GVL.DownDeck1Vis
        tap GVL.DownDeck1
    Polygon (329,357) (335,357) (335,367) (343,367) (343,357) (349,357) (339,347), colour toggle: GVL.UpDeck1Vis
        tap GVL.UpDeck1
    Rectangle (326,297 100x30)
    Rectangle (382,302 20x20), "2"
    Polygon (354,312) (360,312) (360,302) (368,302) (368,312) (374,312) (364,322), colour toggle: GVL.DownDeck2Vis
        tap GVL.DownDeck2
    Polygon (329,312) (335,312) (335,322) (343,322) (343,312) (349,312) (339,302), colour toggle: GVL.UpDeck2Vis
        tap GVL.UpDeck2
    Rectangle (326,250 100x30)
    Rectangle (382,255 20x20), "3"
    Polygon (354,265) (360,265) (360,255) (368,255) (368,265) (374,265) (364,275), colour toggle: GVL.DownDeck3Vis
        tap GVL.DownDeck3
    Polygon (329,265) (335,265) (335,275) (343,275) (343,265) (349,265) (339,255), colour toggle: GVL.UpDeck3Vis
        tap GVL.UpDeck3
    Rectangle (326,204 100x30)
    Rectangle (382,209 20x20), "4"
    Polygon (354,219) (360,219) (360,209) (368,209) (368,219) (374,219) (364,229), colour toggle: GVL.DownDeck4Vis
        tap GVL.DownDeck4
    Polygon (329,219) (335,219) (335,229) (343,229) (343,219) (349,219) (339,209), colour toggle: GVL.UpDeck4Vis
        tap GVL.UpDeck4
    Rectangle (326,158 100x30)
    Rectangle (382,163 20x20), "5"
    Polygon (354,173) (360,173) (360,163) (368,163) (368,173) (374,173) (364,183), colour toggle: GVL.DownDeck5Vis
        tap GVL.DownDeck5
    Polygon (329,173) (335,173) (335,183) (343,183) (343,173) (349,173) (339,163), colour toggle: GVL.UpDeck5Vis
        tap GVL.UpDeck5
    Rectangle (326,113 100x30)
    Rectangle (382,118 20x20), "6"
    Polygon (354,128) (360,128) (360,118) (368,118) (368,128) (374,128) (364,138), colour toggle: GVL.DownDeck6Vis
        tap GVL.DownDeck6
    Polygon (329,128) (335,128) (335,138) (343,138) (343,128) (349,128) (339,118), colour toggle: GVL.UpDeck6Vis
        tap GVL.UpDeck6
    Rectangle (326,68 100x30)
    Rectangle (382,73 20x20), "7"
    Polygon (354,83) (360,83) (360,73) (368,73) (368,83) (374,83) (364,93), colour toggle: GVL.DownDeck7Vis
        tap GVL.DownDeck7
    Rectangle (326,388 100x30)
    Rectangle (382,393 20x20), "G"
    Polygon (329,403) (335,403) (335,413) (343,413) (343,403) (349,403) (339,393), colour toggle: GVL.UpDeckGVis
        tap GVL.UpDeckG
    RoundedRectangle (18,48 100x240)
    Rectangle (18,288 100x20), "Internal Panel"
    Ellipse (74,199 30x30), colour toggle: GVL.P1Vis
    Ellipse (79,204 20x20), "1"
        tap GVL.P1
    Ellipse (32,199 30x30), colour toggle: GVL.PGVis
    Ellipse (37,204 20x20), "G"
        tap GVL.PG
    Ellipse (74,167 30x30), colour toggle: GVL.P3Vis
    Ellipse (79,172 20x20), "3"
        tap GVL.P3
    Ellipse (32,167 30x30), colour toggle: GVL.P2Vis
    Ellipse (37,172 20x20), "2"
        tap GVL.P2
    Ellipse (74,135 30x30), colour toggle: GVL.P5Vis
    Ellipse (79,140 20x20), "5"
        tap GVL.P5
    Ellipse (32,135 30x30), colour toggle: GVL.P4Vis
    Ellipse (37,140 20x20), "4"
        tap GVL.P4
    Ellipse (74,103 30x30), colour toggle: GVL.P7Vis
    Ellipse (79,108 20x20), "7"
        tap GVL.P7
    Ellipse (32,103 30x30), colour toggle: GVL.P6Vis
    Ellipse (37,108 20x20), "6"
        tap GVL.P6
    Rectangle (28,56 80x40), "%s", text variable: GVL.Destination
    Ellipse (43,231 50x50), tooltip "EMERGENCY", colour toggle: GVL.Emergency
    Group (48,236 40x40)
        toggle GVL.Emergency
        Ellipse (0,0 40x40), tooltip "EMERGENCY"
        Polygon (5,28) (10,23) (11,15) (15,8) (20,7) (25,8) (29,15) (30,23) (35,28)
        Ellipse (17,27 6x6)
    Polygon (35,72) (45,62) (55,72), colour toggle: GVL.Motor_on AND GVL.Up
    Polygon (35,80) (45,90) (55,80), colour toggle: GVL.Motor_on AND NOT GVL.Up
    Group (140,48 165x170)
        Rectangle (0,0 165x170)
        Rectangle (15,10 120x160)
        Polygon (40,40) (15,10) (135,10) (110,40)
        Rectangle (40,40 70x100)
        Polygon (15,170) (40,140) (110,140) (135,170)
        Polygon (20,102) (20,53) (35,62) (35,98)
        Polygon (79,35) (79,30) (115,30) (111,35)
        Polygon (39,35) (35,30) (71,30) (71,35)
        Polygon (32,25) (25,15) (70,15) (71,25)
        Polygon (79,25) (80,15) (125,15) (118,25)
        Group (139,82 22x13)
            Rectangle (0,0 22x13)
            Polygon (3,9) (6,4) (9,9)
            Polygon (13,4) (16,9) (19,4)
    BarDisplayImage (410,37 65x412), value: GVL.Height, style: BarDisplayImage-Gray, scale format: %.0f, scale -20..160
        p3451962224: VisuNativeControl.IP_Offline.Browser
    Rectangle (478,68 65x30)
    Rectangle (478,342 65x30)
    Rectangle (478,297 65x30)
    Rectangle (478,250 65x30)
    Rectangle (478,204 65x30)
    Rectangle (478,158 65x30)
    Rectangle (478,113 65x30)
    Rectangle (478,388 65x30)
    RockerSwitch (483,345 19x25), variable: GVL.Ramp1Down, behaviour: TOGGLE, style: Switch-RockerSwitch-Green
    RockerSwitch (503,345 19x25), variable: GVL.Sensor1, behaviour: TOGGLE, style: Switch-RockerSwitch-Red
    RockerSwitch (523,345 19x25), variable: GVL.Ramp1Up, behaviour: TOGGLE, style: Switch-RockerSwitch-Blue
    RockerSwitch (483,300 19x25), variable: GVL.Ramp2Down, behaviour: TOGGLE, style: Switch-RockerSwitch-Green
    RockerSwitch (503,300 19x25), variable: GVL.Sensor2, behaviour: TOGGLE, style: Switch-RockerSwitch-Red
    RockerSwitch (523,300 19x25), variable: GVL.Ramp2Up, behaviour: TOGGLE, style: Switch-RockerSwitch-Blue
    RockerSwitch (483,253 19x25), variable: GVL.Ramp3Down, behaviour: TOGGLE, style: Switch-RockerSwitch-Green
    RockerSwitch (503,253 19x25), variable: GVL.Sensor3, behaviour: TOGGLE, style: Switch-RockerSwitch-Red
    RockerSwitch (523,253 19x25), variable: GVL.Ramp3Up, behaviour: TOGGLE, style: Switch-RockerSwitch-Blue
    RockerSwitch (483,207 19x25), variable: GVL.Ramp4Down, behaviour: TOGGLE, style: Switch-RockerSwitch-Green
    RockerSwitch (503,207 19x25), variable: GVL.Sensor4, behaviour: TOGGLE, style: Switch-RockerSwitch-Red
    RockerSwitch (523,207 19x25), variable: GVL.Ramp4Up, behaviour: TOGGLE, style: Switch-RockerSwitch-Blue
    RockerSwitch (483,161 19x25), variable: GVL.Ramp5Down, behaviour: TOGGLE, style: Switch-RockerSwitch-Green
    RockerSwitch (503,161 19x25), variable: GVL.Sensor5, behaviour: TOGGLE, style: Switch-RockerSwitch-Red
    RockerSwitch (523,161 19x25), variable: GVL.Ramp5Up, behaviour: TOGGLE, style: Switch-RockerSwitch-Blue
    RockerSwitch (483,116 19x25), variable: GVL.Ramp6Down, behaviour: TOGGLE, style: Switch-RockerSwitch-Green
    RockerSwitch (503,116 19x25), variable: GVL.Sensor6, behaviour: TOGGLE, style: Switch-RockerSwitch-Red
    RockerSwitch (523,116 19x25), variable: GVL.Ramp6Up, behaviour: TOGGLE, style: Switch-RockerSwitch-Blue
    RockerSwitch (483,71 19x25), variable: GVL.Ramp7Down, behaviour: TOGGLE, style: Switch-RockerSwitch-Green
    RockerSwitch (503,71 19x25), variable: GVL.Sensor7, behaviour: TOGGLE, style: Switch-RockerSwitch-Red
    RockerSwitch (503,391 19x25), variable: GVL.SensorG, behaviour: TOGGLE, style: Switch-RockerSwitch-Red
    RockerSwitch (523,391 19x25), variable: GVL.RampGUp, behaviour: TOGGLE, style: Switch-RockerSwitch-Blue
    Rectangle (478,28 65x20), "FAULTS"
    Polygon (302,130) (325,113) (326,143) (302,143), invisible if: (GVL.Closing OR GVL.Opening) OR GVL.Closed
    Polygon (118,57) (159,102) (159,151) (119,279), invisible if: (GVL.Closing OR GVL.Opening) OR GVL.Closed
    Rectangle (155,58 0x160)
        p3528305787: GVL.Door
    Rectangle (275,58 0x160)
        p3528305787: -GVL.Door
    Rectangle (23,328 290x20), "System Communications"
    Rectangle (183,353 130x20), "Alarms"
    Rectangle (23,353 75x20), "Deck Sensor", colour toggle: GVL.DeckSensor
    Rectangle (143,378 35x20), "%s", text variable: GVL.Height
    Rectangle (184,388 62x20), "Presence", colour toggle: GVL.Presence
    Rectangle (103,353 75x20), "Ramp Sensor", colour toggle: GVL.RampSensor
    Rectangle (143,403 35x20), "%s", text variable: GVL.Current
    Rectangle (143,428 35x20), "%s", text variable: GVL.Destination
    Rectangle (252,388 62x20), "Deck Fault", colour toggle: GVL.FaultSensorAlarm
    Rectangle (184,418 62x20), "Emergency", colour toggle: GVL.EmergencyVis
    Rectangle (252,418 62x19), "Ramp Fault", colour toggle: GVL.FaultRampAlarm
    Rectangle (23,378 115x20), "Height"
    Rectangle (23,403 115x20), "Current Deck"
    Rectangle (23,428 115x20), "Destination Deck"
    Group (562,25 175x93)
        Rectangle (0,16 175x77)
        Rectangle (7,39 160x30), "This floor sensor"
        Rectangle (7,59 160x30), "Ramp sensor AFTER this floor"
        Rectangle (7,0 70x30), "LEGEND"
        Rectangle (7,20 160x30), "Ramp sensor BEFORE this floor"
    Group (202,232 33x34)
        toggle GVL.Presence
        Rectangle (10,0 8x20)
        Polygon (5,10) (12,20) (14,18) (5,6)
        Ellipse (6,2 5x5)
        Polygon (4,8) (13,12) (14,10) (4,4)
        Rectangle (0,0 8x20)
    Rectangle (169,273 102x31), "Click for presence between the door"
END_VISUALIZATION
